TYPE "LBP_typeTMMagazines"
TITLE = Tool management magazines / Almacenes de gestión de herramientas / Magazine zur Werkzeugverwaltung
// User data type to store the magazine data / Tipo de datos de usuario para guardar los datos de almacén / Anwender-Datentyp zum Speichern der Magazindaten
// stored: IsFailsafeCompliant false
   STRUCT
      MaxSpindleNumber : UInt;   // Maximale Spindelanzahl / Maximum spindle number / Número máximo de cabezales
      NumberOfMagazines : UInt;   // Anzahl aller Magazine einschließlich Belade- und Zwischenspeichermagazine / Number of all magazines including loading and buffer magazines / Número total de almacenes, incluidos almacenes de carga e intermedios
      Magazines : Array[1..64] of Struct   // Alle Magazine einschließlich Belade- und Zwischenspeichermagazine / All magazines including loading and buffer magazines / Todos los almacenes, incluidos almacenes de carga e intermedios
         Number : UInt;   // Magazin-Nummer / Magazine number / Número de almacén
         "Type" : UInt;   // Magazintyp / Magazine type / Tipo de almacén
         Places : UInt;   // Anzahl der Plätze im Magazin / Number of locations in magazine / Número de puestos en el almacén
         TMNumber : UInt;   // Werkzeug-Verwaltungsnummer / Tool management number / Número de gestión de herramientas
      END_STRUCT;
   END_STRUCT;
   // // Magazines[2].Number : Magazin-Nummer / Magazine number / Número de almacén
   // // Magazines[3].Number : Magazin-Nummer / Magazine number / Número de almacén
   // // Magazines[4].Number : Magazin-Nummer / Magazine number / Número de almacén
   // // Magazines[5].Number : Magazin-Nummer / Magazine number / Número de almacén
   // // Magazines[6].Number : Magazin-Nummer / Magazine number / Número de almacén
   // // Magazines[7].Number : Magazin-Nummer / Magazine number / Número de almacén
   // // Magazines[8].Number : Magazin-Nummer / Magazine number / Número de almacén
   // // Magazines[9].Number : Magazin-Nummer / Magazine number / Número de almacén
   // // Magazines[10].Number : Magazin-Nummer / Magazine number / Número de almacén
   // // Magazines[11].Number : Magazin-Nummer / Magazine number / Número de almacén
   // // Magazines[12].Number : Magazin-Nummer / Magazine number / Número de almacén
   // // Magazines[13].Number : Magazin-Nummer / Magazine number / Número de almacén
   // // Magazines[14].Number : Magazin-Nummer / Magazine number / Número de almacén
   // // Magazines[15].Number : Magazin-Nummer / Magazine number / Número de almacén
   // // Magazines[16].Number : Magazin-Nummer / Magazine number / Número de almacén
   // // Magazines[17].Number : Magazin-Nummer / Magazine number / Número de almacén
   // // Magazines[18].Number : Magazin-Nummer / Magazine number / Número de almacén
   // // Magazines[19].Number : Magazin-Nummer / Magazine number / Número de almacén
   // // Magazines[20].Number : Magazin-Nummer / Magazine number / Número de almacén
   // // Magazines[21].Number : Magazin-Nummer / Magazine number / Número de almacén
   // // Magazines[22].Number : Magazin-Nummer / Magazine number / Número de almacén
   // // Magazines[23].Number : Magazin-Nummer / Magazine number / Número de almacén
   // // Magazines[24].Number : Magazin-Nummer / Magazine number / Número de almacén
   // // Magazines[25].Number : Magazin-Nummer / Magazine number / Número de almacén
   // // Magazines[26].Number : Magazin-Nummer / Magazine number / Número de almacén
   // // Magazines[27].Number : Magazin-Nummer / Magazine number / Número de almacén
   // // Magazines[28].Number : Magazin-Nummer / Magazine number / Número de almacén
   // // Magazines[29].Number : Magazin-Nummer / Magazine number / Número de almacén
   // // Magazines[30].Number : Magazin-Nummer / Magazine number / Número de almacén
   // // Magazines[31].Number : Magazin-Nummer / Magazine number / Número de almacén
   // // Magazines[32].Number : Magazin-Nummer / Magazine number / Número de almacén
   // // Magazines[33].Number : Magazin-Nummer / Magazine number / Número de almacén
   // // Magazines[34].Number : Magazin-Nummer / Magazine number / Número de almacén
   // // Magazines[35].Number : Magazin-Nummer / Magazine number / Número de almacén
   // // Magazines[36].Number : Magazin-Nummer / Magazine number / Número de almacén
   // // Magazines[37].Number : Magazin-Nummer / Magazine number / Número de almacén
   // // Magazines[38].Number : Magazin-Nummer / Magazine number / Número de almacén
   // // Magazines[39].Number : Magazin-Nummer / Magazine number / Número de almacén
   // // Magazines[40].Number : Magazin-Nummer / Magazine number / Número de almacén
   // // Magazines[41].Number : Magazin-Nummer / Magazine number / Número de almacén
   // // Magazines[42].Number : Magazin-Nummer / Magazine number / Número de almacén
   // // Magazines[43].Number : Magazin-Nummer / Magazine number / Número de almacén
   // // Magazines[44].Number : Magazin-Nummer / Magazine number / Número de almacén
   // // Magazines[45].Number : Magazin-Nummer / Magazine number / Número de almacén
   // // Magazines[46].Number : Magazin-Nummer / Magazine number / Número de almacén
   // // Magazines[47].Number : Magazin-Nummer / Magazine number / Número de almacén
   // // Magazines[48].Number : Magazin-Nummer / Magazine number / Número de almacén
   // // Magazines[49].Number : Magazin-Nummer / Magazine number / Número de almacén
   // // Magazines[50].Number : Magazin-Nummer / Magazine number / Número de almacén
   // // Magazines[51].Number : Magazin-Nummer / Magazine number / Número de almacén
   // // Magazines[52].Number : Magazin-Nummer / Magazine number / Número de almacén
   // // Magazines[53].Number : Magazin-Nummer / Magazine number / Número de almacén
   // // Magazines[54].Number : Magazin-Nummer / Magazine number / Número de almacén
   // // Magazines[55].Number : Magazin-Nummer / Magazine number / Número de almacén
   // // Magazines[56].Number : Magazin-Nummer / Magazine number / Número de almacén
   // // Magazines[57].Number : Magazin-Nummer / Magazine number / Número de almacén
   // // Magazines[58].Number : Magazin-Nummer / Magazine number / Número de almacén
   // // Magazines[59].Number : Magazin-Nummer / Magazine number / Número de almacén
   // // Magazines[60].Number : Magazin-Nummer / Magazine number / Número de almacén
   // // Magazines[61].Number : Magazin-Nummer / Magazine number / Número de almacén
   // // Magazines[62].Number : Magazin-Nummer / Magazine number / Número de almacén
   // // Magazines[63].Number : Magazin-Nummer / Magazine number / Número de almacén
   // // Magazines[64].Number : Magazin-Nummer / Magazine number / Número de almacén
   // // Magazines[2]."Type" : Magazintyp / Magazine type / Tipo de almacén
   // // Magazines[3]."Type" : Magazintyp / Magazine type / Tipo de almacén
   // // Magazines[4]."Type" : Magazintyp / Magazine type / Tipo de almacén
   // // Magazines[5]."Type" : Magazintyp / Magazine type / Tipo de almacén
   // // Magazines[6]."Type" : Magazintyp / Magazine type / Tipo de almacén
   // // Magazines[7]."Type" : Magazintyp / Magazine type / Tipo de almacén
   // // Magazines[8]."Type" : Magazintyp / Magazine type / Tipo de almacén
   // // Magazines[9]."Type" : Magazintyp / Magazine type / Tipo de almacén
   // // Magazines[10]."Type" : Magazintyp / Magazine type / Tipo de almacén
   // // Magazines[11]."Type" : Magazintyp / Magazine type / Tipo de almacén
   // // Magazines[12]."Type" : Magazintyp / Magazine type / Tipo de almacén
   // // Magazines[13]."Type" : Magazintyp / Magazine type / Tipo de almacén
   // // Magazines[14]."Type" : Magazintyp / Magazine type / Tipo de almacén
   // // Magazines[15]."Type" : Magazintyp / Magazine type / Tipo de almacén
   // // Magazines[16]."Type" : Magazintyp / Magazine type / Tipo de almacén
   // // Magazines[17]."Type" : Magazintyp / Magazine type / Tipo de almacén
   // // Magazines[18]."Type" : Magazintyp / Magazine type / Tipo de almacén
   // // Magazines[19]."Type" : Magazintyp / Magazine type / Tipo de almacén
   // // Magazines[20]."Type" : Magazintyp / Magazine type / Tipo de almacén
   // // Magazines[21]."Type" : Magazintyp / Magazine type / Tipo de almacén
   // // Magazines[22]."Type" : Magazintyp / Magazine type / Tipo de almacén
   // // Magazines[23]."Type" : Magazintyp / Magazine type / Tipo de almacén
   // // Magazines[24]."Type" : Magazintyp / Magazine type / Tipo de almacén
   // // Magazines[25]."Type" : Magazintyp / Magazine type / Tipo de almacén
   // // Magazines[26]."Type" : Magazintyp / Magazine type / Tipo de almacén
   // // Magazines[27]."Type" : Magazintyp / Magazine type / Tipo de almacén
   // // Magazines[28]."Type" : Magazintyp / Magazine type / Tipo de almacén
   // // Magazines[29]."Type" : Magazintyp / Magazine type / Tipo de almacén
   // // Magazines[30]."Type" : Magazintyp / Magazine type / Tipo de almacén
   // // Magazines[31]."Type" : Magazintyp / Magazine type / Tipo de almacén
   // // Magazines[32]."Type" : Magazintyp / Magazine type / Tipo de almacén
   // // Magazines[33]."Type" : Magazintyp / Magazine type / Tipo de almacén
   // // Magazines[34]."Type" : Magazintyp / Magazine type / Tipo de almacén
   // // Magazines[35]."Type" : Magazintyp / Magazine type / Tipo de almacén
   // // Magazines[36]."Type" : Magazintyp / Magazine type / Tipo de almacén
   // // Magazines[37]."Type" : Magazintyp / Magazine type / Tipo de almacén
   // // Magazines[38]."Type" : Magazintyp / Magazine type / Tipo de almacén
   // // Magazines[39]."Type" : Magazintyp / Magazine type / Tipo de almacén
   // // Magazines[40]."Type" : Magazintyp / Magazine type / Tipo de almacén
   // // Magazines[41]."Type" : Magazintyp / Magazine type / Tipo de almacén
   // // Magazines[42]."Type" : Magazintyp / Magazine type / Tipo de almacén
   // // Magazines[43]."Type" : Magazintyp / Magazine type / Tipo de almacén
   // // Magazines[44]."Type" : Magazintyp / Magazine type / Tipo de almacén
   // // Magazines[45]."Type" : Magazintyp / Magazine type / Tipo de almacén
   // // Magazines[46]."Type" : Magazintyp / Magazine type / Tipo de almacén
   // // Magazines[47]."Type" : Magazintyp / Magazine type / Tipo de almacén
   // // Magazines[48]."Type" : Magazintyp / Magazine type / Tipo de almacén
   // // Magazines[49]."Type" : Magazintyp / Magazine type / Tipo de almacén
   // // Magazines[50]."Type" : Magazintyp / Magazine type / Tipo de almacén
   // // Magazines[51]."Type" : Magazintyp / Magazine type / Tipo de almacén
   // // Magazines[52]."Type" : Magazintyp / Magazine type / Tipo de almacén
   // // Magazines[53]."Type" : Magazintyp / Magazine type / Tipo de almacén
   // // Magazines[54]."Type" : Magazintyp / Magazine type / Tipo de almacén
   // // Magazines[55]."Type" : Magazintyp / Magazine type / Tipo de almacén
   // // Magazines[56]."Type" : Magazintyp / Magazine type / Tipo de almacén
   // // Magazines[57]."Type" : Magazintyp / Magazine type / Tipo de almacén
   // // Magazines[58]."Type" : Magazintyp / Magazine type / Tipo de almacén
   // // Magazines[59]."Type" : Magazintyp / Magazine type / Tipo de almacén
   // // Magazines[60]."Type" : Magazintyp / Magazine type / Tipo de almacén
   // // Magazines[61]."Type" : Magazintyp / Magazine type / Tipo de almacén
   // // Magazines[62]."Type" : Magazintyp / Magazine type / Tipo de almacén
   // // Magazines[63]."Type" : Magazintyp / Magazine type / Tipo de almacén
   // // Magazines[64]."Type" : Magazintyp / Magazine type / Tipo de almacén
   // // Magazines[2].Places : Anzahl der Plätze im Magazin / Number of locations in magazine / Número de puestos en el almacén
   // // Magazines[3].Places : Anzahl der Plätze im Magazin / Number of locations in magazine / Número de puestos en el almacén
   // // Magazines[4].Places : Anzahl der Plätze im Magazin / Number of locations in magazine / Número de puestos en el almacén
   // // Magazines[5].Places : Anzahl der Plätze im Magazin / Number of locations in magazine / Número de puestos en el almacén
   // // Magazines[6].Places : Anzahl der Plätze im Magazin / Number of locations in magazine / Número de puestos en el almacén
   // // Magazines[7].Places : Anzahl der Plätze im Magazin / Number of locations in magazine / Número de puestos en el almacén
   // // Magazines[8].Places : Anzahl der Plätze im Magazin / Number of locations in magazine / Número de puestos en el almacén
   // // Magazines[9].Places : Anzahl der Plätze im Magazin / Number of locations in magazine / Número de puestos en el almacén
   // // Magazines[10].Places : Anzahl der Plätze im Magazin / Number of locations in magazine / Número de puestos en el almacén
   // // Magazines[11].Places : Anzahl der Plätze im Magazin / Number of locations in magazine / Número de puestos en el almacén
   // // Magazines[12].Places : Anzahl der Plätze im Magazin / Number of locations in magazine / Número de puestos en el almacén
   // // Magazines[13].Places : Anzahl der Plätze im Magazin / Number of locations in magazine / Número de puestos en el almacén
   // // Magazines[14].Places : Anzahl der Plätze im Magazin / Number of locations in magazine / Número de puestos en el almacén
   // // Magazines[15].Places : Anzahl der Plätze im Magazin / Number of locations in magazine / Número de puestos en el almacén
   // // Magazines[16].Places : Anzahl der Plätze im Magazin / Number of locations in magazine / Número de puestos en el almacén
   // // Magazines[17].Places : Anzahl der Plätze im Magazin / Number of locations in magazine / Número de puestos en el almacén
   // // Magazines[18].Places : Anzahl der Plätze im Magazin / Number of locations in magazine / Número de puestos en el almacén
   // // Magazines[19].Places : Anzahl der Plätze im Magazin / Number of locations in magazine / Número de puestos en el almacén
   // // Magazines[20].Places : Anzahl der Plätze im Magazin / Number of locations in magazine / Número de puestos en el almacén
   // // Magazines[21].Places : Anzahl der Plätze im Magazin / Number of locations in magazine / Número de puestos en el almacén
   // // Magazines[22].Places : Anzahl der Plätze im Magazin / Number of locations in magazine / Número de puestos en el almacén
   // // Magazines[23].Places : Anzahl der Plätze im Magazin / Number of locations in magazine / Número de puestos en el almacén
   // // Magazines[24].Places : Anzahl der Plätze im Magazin / Number of locations in magazine / Número de puestos en el almacén
   // // Magazines[25].Places : Anzahl der Plätze im Magazin / Number of locations in magazine / Número de puestos en el almacén
   // // Magazines[26].Places : Anzahl der Plätze im Magazin / Number of locations in magazine / Número de puestos en el almacén
   // // Magazines[27].Places : Anzahl der Plätze im Magazin / Number of locations in magazine / Número de puestos en el almacén
   // // Magazines[28].Places : Anzahl der Plätze im Magazin / Number of locations in magazine / Número de puestos en el almacén
   // // Magazines[29].Places : Anzahl der Plätze im Magazin / Number of locations in magazine / Número de puestos en el almacén
   // // Magazines[30].Places : Anzahl der Plätze im Magazin / Number of locations in magazine / Número de puestos en el almacén
   // // Magazines[31].Places : Anzahl der Plätze im Magazin / Number of locations in magazine / Número de puestos en el almacén
   // // Magazines[32].Places : Anzahl der Plätze im Magazin / Number of locations in magazine / Número de puestos en el almacén
   // // Magazines[33].Places : Anzahl der Plätze im Magazin / Number of locations in magazine / Número de puestos en el almacén
   // // Magazines[34].Places : Anzahl der Plätze im Magazin / Number of locations in magazine / Número de puestos en el almacén
   // // Magazines[35].Places : Anzahl der Plätze im Magazin / Number of locations in magazine / Número de puestos en el almacén
   // // Magazines[36].Places : Anzahl der Plätze im Magazin / Number of locations in magazine / Número de puestos en el almacén
   // // Magazines[37].Places : Anzahl der Plätze im Magazin / Number of locations in magazine / Número de puestos en el almacén
   // // Magazines[38].Places : Anzahl der Plätze im Magazin / Number of locations in magazine / Número de puestos en el almacén
   // // Magazines[39].Places : Anzahl der Plätze im Magazin / Number of locations in magazine / Número de puestos en el almacén
   // // Magazines[40].Places : Anzahl der Plätze im Magazin / Number of locations in magazine / Número de puestos en el almacén
   // // Magazines[41].Places : Anzahl der Plätze im Magazin / Number of locations in magazine / Número de puestos en el almacén
   // // Magazines[42].Places : Anzahl der Plätze im Magazin / Number of locations in magazine / Número de puestos en el almacén
   // // Magazines[43].Places : Anzahl der Plätze im Magazin / Number of locations in magazine / Número de puestos en el almacén
   // // Magazines[44].Places : Anzahl der Plätze im Magazin / Number of locations in magazine / Número de puestos en el almacén
   // // Magazines[45].Places : Anzahl der Plätze im Magazin / Number of locations in magazine / Número de puestos en el almacén
   // // Magazines[46].Places : Anzahl der Plätze im Magazin / Number of locations in magazine / Número de puestos en el almacén
   // // Magazines[47].Places : Anzahl der Plätze im Magazin / Number of locations in magazine / Número de puestos en el almacén
   // // Magazines[48].Places : Anzahl der Plätze im Magazin / Number of locations in magazine / Número de puestos en el almacén
   // // Magazines[49].Places : Anzahl der Plätze im Magazin / Number of locations in magazine / Número de puestos en el almacén
   // // Magazines[50].Places : Anzahl der Plätze im Magazin / Number of locations in magazine / Número de puestos en el almacén
   // // Magazines[51].Places : Anzahl der Plätze im Magazin / Number of locations in magazine / Número de puestos en el almacén
   // // Magazines[52].Places : Anzahl der Plätze im Magazin / Number of locations in magazine / Número de puestos en el almacén
   // // Magazines[53].Places : Anzahl der Plätze im Magazin / Number of locations in magazine / Número de puestos en el almacén
   // // Magazines[54].Places : Anzahl der Plätze im Magazin / Number of locations in magazine / Número de puestos en el almacén
   // // Magazines[55].Places : Anzahl der Plätze im Magazin / Number of locations in magazine / Número de puestos en el almacén
   // // Magazines[56].Places : Anzahl der Plätze im Magazin / Number of locations in magazine / Número de puestos en el almacén
   // // Magazines[57].Places : Anzahl der Plätze im Magazin / Number of locations in magazine / Número de puestos en el almacén
   // // Magazines[58].Places : Anzahl der Plätze im Magazin / Number of locations in magazine / Número de puestos en el almacén
   // // Magazines[59].Places : Anzahl der Plätze im Magazin / Number of locations in magazine / Número de puestos en el almacén
   // // Magazines[60].Places : Anzahl der Plätze im Magazin / Number of locations in magazine / Número de puestos en el almacén
   // // Magazines[61].Places : Anzahl der Plätze im Magazin / Number of locations in magazine / Número de puestos en el almacén
   // // Magazines[62].Places : Anzahl der Plätze im Magazin / Number of locations in magazine / Número de puestos en el almacén
   // // Magazines[63].Places : Anzahl der Plätze im Magazin / Number of locations in magazine / Número de puestos en el almacén
   // // Magazines[64].Places : Anzahl der Plätze im Magazin / Number of locations in magazine / Número de puestos en el almacén
   // // Magazines[2].TMNumber : Werkzeug-Verwaltungsnummer / Tool management number / Número de gestión de herramientas
   // // Magazines[3].TMNumber : Werkzeug-Verwaltungsnummer / Tool management number / Número de gestión de herramientas
   // // Magazines[4].TMNumber : Werkzeug-Verwaltungsnummer / Tool management number / Número de gestión de herramientas
   // // Magazines[5].TMNumber : Werkzeug-Verwaltungsnummer / Tool management number / Número de gestión de herramientas
   // // Magazines[6].TMNumber : Werkzeug-Verwaltungsnummer / Tool management number / Número de gestión de herramientas
   // // Magazines[7].TMNumber : Werkzeug-Verwaltungsnummer / Tool management number / Número de gestión de herramientas
   // // Magazines[8].TMNumber : Werkzeug-Verwaltungsnummer / Tool management number / Número de gestión de herramientas
   // // Magazines[9].TMNumber : Werkzeug-Verwaltungsnummer / Tool management number / Número de gestión de herramientas
   // // Magazines[10].TMNumber : Werkzeug-Verwaltungsnummer / Tool management number / Número de gestión de herramientas
   // // Magazines[11].TMNumber : Werkzeug-Verwaltungsnummer / Tool management number / Número de gestión de herramientas
   // // Magazines[12].TMNumber : Werkzeug-Verwaltungsnummer / Tool management number / Número de gestión de herramientas
   // // Magazines[13].TMNumber : Werkzeug-Verwaltungsnummer / Tool management number / Número de gestión de herramientas
   // // Magazines[14].TMNumber : Werkzeug-Verwaltungsnummer / Tool management number / Número de gestión de herramientas
   // // Magazines[15].TMNumber : Werkzeug-Verwaltungsnummer / Tool management number / Número de gestión de herramientas
   // // Magazines[16].TMNumber : Werkzeug-Verwaltungsnummer / Tool management number / Número de gestión de herramientas
   // // Magazines[17].TMNumber : Werkzeug-Verwaltungsnummer / Tool management number / Número de gestión de herramientas
   // // Magazines[18].TMNumber : Werkzeug-Verwaltungsnummer / Tool management number / Número de gestión de herramientas
   // // Magazines[19].TMNumber : Werkzeug-Verwaltungsnummer / Tool management number / Número de gestión de herramientas
   // // Magazines[20].TMNumber : Werkzeug-Verwaltungsnummer / Tool management number / Número de gestión de herramientas
   // // Magazines[21].TMNumber : Werkzeug-Verwaltungsnummer / Tool management number / Número de gestión de herramientas
   // // Magazines[22].TMNumber : Werkzeug-Verwaltungsnummer / Tool management number / Número de gestión de herramientas
   // // Magazines[23].TMNumber : Werkzeug-Verwaltungsnummer / Tool management number / Número de gestión de herramientas
   // // Magazines[24].TMNumber : Werkzeug-Verwaltungsnummer / Tool management number / Número de gestión de herramientas
   // // Magazines[25].TMNumber : Werkzeug-Verwaltungsnummer / Tool management number / Número de gestión de herramientas
   // // Magazines[26].TMNumber : Werkzeug-Verwaltungsnummer / Tool management number / Número de gestión de herramientas
   // // Magazines[27].TMNumber : Werkzeug-Verwaltungsnummer / Tool management number / Número de gestión de herramientas
   // // Magazines[28].TMNumber : Werkzeug-Verwaltungsnummer / Tool management number / Número de gestión de herramientas
   // // Magazines[29].TMNumber : Werkzeug-Verwaltungsnummer / Tool management number / Número de gestión de herramientas
   // // Magazines[30].TMNumber : Werkzeug-Verwaltungsnummer / Tool management number / Número de gestión de herramientas
   // // Magazines[31].TMNumber : Werkzeug-Verwaltungsnummer / Tool management number / Número de gestión de herramientas
   // // Magazines[32].TMNumber : Werkzeug-Verwaltungsnummer / Tool management number / Número de gestión de herramientas
   // // Magazines[33].TMNumber : Werkzeug-Verwaltungsnummer / Tool management number / Número de gestión de herramientas
   // // Magazines[34].TMNumber : Werkzeug-Verwaltungsnummer / Tool management number / Número de gestión de herramientas
   // // Magazines[35].TMNumber : Werkzeug-Verwaltungsnummer / Tool management number / Número de gestión de herramientas
   // // Magazines[36].TMNumber : Werkzeug-Verwaltungsnummer / Tool management number / Número de gestión de herramientas
   // // Magazines[37].TMNumber : Werkzeug-Verwaltungsnummer / Tool management number / Número de gestión de herramientas
   // // Magazines[38].TMNumber : Werkzeug-Verwaltungsnummer / Tool management number / Número de gestión de herramientas
   // // Magazines[39].TMNumber : Werkzeug-Verwaltungsnummer / Tool management number / Número de gestión de herramientas
   // // Magazines[40].TMNumber : Werkzeug-Verwaltungsnummer / Tool management number / Número de gestión de herramientas
   // // Magazines[41].TMNumber : Werkzeug-Verwaltungsnummer / Tool management number / Número de gestión de herramientas
   // // Magazines[42].TMNumber : Werkzeug-Verwaltungsnummer / Tool management number / Número de gestión de herramientas
   // // Magazines[43].TMNumber : Werkzeug-Verwaltungsnummer / Tool management number / Número de gestión de herramientas
   // // Magazines[44].TMNumber : Werkzeug-Verwaltungsnummer / Tool management number / Número de gestión de herramientas
   // // Magazines[45].TMNumber : Werkzeug-Verwaltungsnummer / Tool management number / Número de gestión de herramientas
   // // Magazines[46].TMNumber : Werkzeug-Verwaltungsnummer / Tool management number / Número de gestión de herramientas
   // // Magazines[47].TMNumber : Werkzeug-Verwaltungsnummer / Tool management number / Número de gestión de herramientas
   // // Magazines[48].TMNumber : Werkzeug-Verwaltungsnummer / Tool management number / Número de gestión de herramientas
   // // Magazines[49].TMNumber : Werkzeug-Verwaltungsnummer / Tool management number / Número de gestión de herramientas
   // // Magazines[50].TMNumber : Werkzeug-Verwaltungsnummer / Tool management number / Número de gestión de herramientas
   // // Magazines[51].TMNumber : Werkzeug-Verwaltungsnummer / Tool management number / Número de gestión de herramientas
   // // Magazines[52].TMNumber : Werkzeug-Verwaltungsnummer / Tool management number / Número de gestión de herramientas
   // // Magazines[53].TMNumber : Werkzeug-Verwaltungsnummer / Tool management number / Número de gestión de herramientas
   // // Magazines[54].TMNumber : Werkzeug-Verwaltungsnummer / Tool management number / Número de gestión de herramientas
   // // Magazines[55].TMNumber : Werkzeug-Verwaltungsnummer / Tool management number / Número de gestión de herramientas
   // // Magazines[56].TMNumber : Werkzeug-Verwaltungsnummer / Tool management number / Número de gestión de herramientas
   // // Magazines[57].TMNumber : Werkzeug-Verwaltungsnummer / Tool management number / Número de gestión de herramientas
   // // Magazines[58].TMNumber : Werkzeug-Verwaltungsnummer / Tool management number / Número de gestión de herramientas
   // // Magazines[59].TMNumber : Werkzeug-Verwaltungsnummer / Tool management number / Número de gestión de herramientas
   // // Magazines[60].TMNumber : Werkzeug-Verwaltungsnummer / Tool management number / Número de gestión de herramientas
   // // Magazines[61].TMNumber : Werkzeug-Verwaltungsnummer / Tool management number / Número de gestión de herramientas
   // // Magazines[62].TMNumber : Werkzeug-Verwaltungsnummer / Tool management number / Número de gestión de herramientas
   // // Magazines[63].TMNumber : Werkzeug-Verwaltungsnummer / Tool management number / Número de gestión de herramientas
   // // Magazines[64].TMNumber : Werkzeug-Verwaltungsnummer / Tool management number / Número de gestión de herramientas
   // // Magazines[1] : Alle Magazine einschließlich Belade- und Zwischenspeichermagazine / All magazines including loading and buffer magazines / Todos los almacenes, incluidos almacenes de carga e intermedios
   // // Magazines[2] : Alle Magazine einschließlich Belade- und Zwischenspeichermagazine / All magazines including loading and buffer magazines / Todos los almacenes, incluidos almacenes de carga e intermedios
   // // Magazines[3] : Alle Magazine einschließlich Belade- und Zwischenspeichermagazine / All magazines including loading and buffer magazines / Todos los almacenes, incluidos almacenes de carga e intermedios
   // // Magazines[4] : Alle Magazine einschließlich Belade- und Zwischenspeichermagazine / All magazines including loading and buffer magazines / Todos los almacenes, incluidos almacenes de carga e intermedios
   // // Magazines[5] : Alle Magazine einschließlich Belade- und Zwischenspeichermagazine / All magazines including loading and buffer magazines / Todos los almacenes, incluidos almacenes de carga e intermedios
   // // Magazines[6] : Alle Magazine einschließlich Belade- und Zwischenspeichermagazine / All magazines including loading and buffer magazines / Todos los almacenes, incluidos almacenes de carga e intermedios
   // // Magazines[7] : Alle Magazine einschließlich Belade- und Zwischenspeichermagazine / All magazines including loading and buffer magazines / Todos los almacenes, incluidos almacenes de carga e intermedios
   // // Magazines[8] : Alle Magazine einschließlich Belade- und Zwischenspeichermagazine / All magazines including loading and buffer magazines / Todos los almacenes, incluidos almacenes de carga e intermedios
   // // Magazines[9] : Alle Magazine einschließlich Belade- und Zwischenspeichermagazine / All magazines including loading and buffer magazines / Todos los almacenes, incluidos almacenes de carga e intermedios
   // // Magazines[10] : Alle Magazine einschließlich Belade- und Zwischenspeichermagazine / All magazines including loading and buffer magazines / Todos los almacenes, incluidos almacenes de carga e intermedios
   // // Magazines[11] : Alle Magazine einschließlich Belade- und Zwischenspeichermagazine / All magazines including loading and buffer magazines / Todos los almacenes, incluidos almacenes de carga e intermedios
   // // Magazines[12] : Alle Magazine einschließlich Belade- und Zwischenspeichermagazine / All magazines including loading and buffer magazines / Todos los almacenes, incluidos almacenes de carga e intermedios
   // // Magazines[13] : Alle Magazine einschließlich Belade- und Zwischenspeichermagazine / All magazines including loading and buffer magazines / Todos los almacenes, incluidos almacenes de carga e intermedios
   // // Magazines[14] : Alle Magazine einschließlich Belade- und Zwischenspeichermagazine / All magazines including loading and buffer magazines / Todos los almacenes, incluidos almacenes de carga e intermedios
   // // Magazines[15] : Alle Magazine einschließlich Belade- und Zwischenspeichermagazine / All magazines including loading and buffer magazines / Todos los almacenes, incluidos almacenes de carga e intermedios
   // // Magazines[16] : Alle Magazine einschließlich Belade- und Zwischenspeichermagazine / All magazines including loading and buffer magazines / Todos los almacenes, incluidos almacenes de carga e intermedios
   // // Magazines[17] : Alle Magazine einschließlich Belade- und Zwischenspeichermagazine / All magazines including loading and buffer magazines / Todos los almacenes, incluidos almacenes de carga e intermedios
   // // Magazines[18] : Alle Magazine einschließlich Belade- und Zwischenspeichermagazine / All magazines including loading and buffer magazines / Todos los almacenes, incluidos almacenes de carga e intermedios
   // // Magazines[19] : Alle Magazine einschließlich Belade- und Zwischenspeichermagazine / All magazines including loading and buffer magazines / Todos los almacenes, incluidos almacenes de carga e intermedios
   // // Magazines[20] : Alle Magazine einschließlich Belade- und Zwischenspeichermagazine / All magazines including loading and buffer magazines / Todos los almacenes, incluidos almacenes de carga e intermedios
   // // Magazines[21] : Alle Magazine einschließlich Belade- und Zwischenspeichermagazine / All magazines including loading and buffer magazines / Todos los almacenes, incluidos almacenes de carga e intermedios
   // // Magazines[22] : Alle Magazine einschließlich Belade- und Zwischenspeichermagazine / All magazines including loading and buffer magazines / Todos los almacenes, incluidos almacenes de carga e intermedios
   // // Magazines[23] : Alle Magazine einschließlich Belade- und Zwischenspeichermagazine / All magazines including loading and buffer magazines / Todos los almacenes, incluidos almacenes de carga e intermedios
   // // Magazines[24] : Alle Magazine einschließlich Belade- und Zwischenspeichermagazine / All magazines including loading and buffer magazines / Todos los almacenes, incluidos almacenes de carga e intermedios
   // // Magazines[25] : Alle Magazine einschließlich Belade- und Zwischenspeichermagazine / All magazines including loading and buffer magazines / Todos los almacenes, incluidos almacenes de carga e intermedios
   // // Magazines[26] : Alle Magazine einschließlich Belade- und Zwischenspeichermagazine / All magazines including loading and buffer magazines / Todos los almacenes, incluidos almacenes de carga e intermedios
   // // Magazines[27] : Alle Magazine einschließlich Belade- und Zwischenspeichermagazine / All magazines including loading and buffer magazines / Todos los almacenes, incluidos almacenes de carga e intermedios
   // // Magazines[28] : Alle Magazine einschließlich Belade- und Zwischenspeichermagazine / All magazines including loading and buffer magazines / Todos los almacenes, incluidos almacenes de carga e intermedios
   // // Magazines[29] : Alle Magazine einschließlich Belade- und Zwischenspeichermagazine / All magazines including loading and buffer magazines / Todos los almacenes, incluidos almacenes de carga e intermedios
   // // Magazines[30] : Alle Magazine einschließlich Belade- und Zwischenspeichermagazine / All magazines including loading and buffer magazines / Todos los almacenes, incluidos almacenes de carga e intermedios
   // // Magazines[31] : Alle Magazine einschließlich Belade- und Zwischenspeichermagazine / All magazines including loading and buffer magazines / Todos los almacenes, incluidos almacenes de carga e intermedios
   // // Magazines[32] : Alle Magazine einschließlich Belade- und Zwischenspeichermagazine / All magazines including loading and buffer magazines / Todos los almacenes, incluidos almacenes de carga e intermedios
   // // Magazines[33] : Alle Magazine einschließlich Belade- und Zwischenspeichermagazine / All magazines including loading and buffer magazines / Todos los almacenes, incluidos almacenes de carga e intermedios
   // // Magazines[34] : Alle Magazine einschließlich Belade- und Zwischenspeichermagazine / All magazines including loading and buffer magazines / Todos los almacenes, incluidos almacenes de carga e intermedios
   // // Magazines[35] : Alle Magazine einschließlich Belade- und Zwischenspeichermagazine / All magazines including loading and buffer magazines / Todos los almacenes, incluidos almacenes de carga e intermedios
   // // Magazines[36] : Alle Magazine einschließlich Belade- und Zwischenspeichermagazine / All magazines including loading and buffer magazines / Todos los almacenes, incluidos almacenes de carga e intermedios
   // // Magazines[37] : Alle Magazine einschließlich Belade- und Zwischenspeichermagazine / All magazines including loading and buffer magazines / Todos los almacenes, incluidos almacenes de carga e intermedios
   // // Magazines[38] : Alle Magazine einschließlich Belade- und Zwischenspeichermagazine / All magazines including loading and buffer magazines / Todos los almacenes, incluidos almacenes de carga e intermedios
   // // Magazines[39] : Alle Magazine einschließlich Belade- und Zwischenspeichermagazine / All magazines including loading and buffer magazines / Todos los almacenes, incluidos almacenes de carga e intermedios
   // // Magazines[40] : Alle Magazine einschließlich Belade- und Zwischenspeichermagazine / All magazines including loading and buffer magazines / Todos los almacenes, incluidos almacenes de carga e intermedios
   // // Magazines[41] : Alle Magazine einschließlich Belade- und Zwischenspeichermagazine / All magazines including loading and buffer magazines / Todos los almacenes, incluidos almacenes de carga e intermedios
   // // Magazines[42] : Alle Magazine einschließlich Belade- und Zwischenspeichermagazine / All magazines including loading and buffer magazines / Todos los almacenes, incluidos almacenes de carga e intermedios
   // // Magazines[43] : Alle Magazine einschließlich Belade- und Zwischenspeichermagazine / All magazines including loading and buffer magazines / Todos los almacenes, incluidos almacenes de carga e intermedios
   // // Magazines[44] : Alle Magazine einschließlich Belade- und Zwischenspeichermagazine / All magazines including loading and buffer magazines / Todos los almacenes, incluidos almacenes de carga e intermedios
   // // Magazines[45] : Alle Magazine einschließlich Belade- und Zwischenspeichermagazine / All magazines including loading and buffer magazines / Todos los almacenes, incluidos almacenes de carga e intermedios
   // // Magazines[46] : Alle Magazine einschließlich Belade- und Zwischenspeichermagazine / All magazines including loading and buffer magazines / Todos los almacenes, incluidos almacenes de carga e intermedios
   // // Magazines[47] : Alle Magazine einschließlich Belade- und Zwischenspeichermagazine / All magazines including loading and buffer magazines / Todos los almacenes, incluidos almacenes de carga e intermedios
   // // Magazines[48] : Alle Magazine einschließlich Belade- und Zwischenspeichermagazine / All magazines including loading and buffer magazines / Todos los almacenes, incluidos almacenes de carga e intermedios
   // // Magazines[49] : Alle Magazine einschließlich Belade- und Zwischenspeichermagazine / All magazines including loading and buffer magazines / Todos los almacenes, incluidos almacenes de carga e intermedios
   // // Magazines[50] : Alle Magazine einschließlich Belade- und Zwischenspeichermagazine / All magazines including loading and buffer magazines / Todos los almacenes, incluidos almacenes de carga e intermedios
   // // Magazines[51] : Alle Magazine einschließlich Belade- und Zwischenspeichermagazine / All magazines including loading and buffer magazines / Todos los almacenes, incluidos almacenes de carga e intermedios
   // // Magazines[52] : Alle Magazine einschließlich Belade- und Zwischenspeichermagazine / All magazines including loading and buffer magazines / Todos los almacenes, incluidos almacenes de carga e intermedios
   // // Magazines[53] : Alle Magazine einschließlich Belade- und Zwischenspeichermagazine / All magazines including loading and buffer magazines / Todos los almacenes, incluidos almacenes de carga e intermedios
   // // Magazines[54] : Alle Magazine einschließlich Belade- und Zwischenspeichermagazine / All magazines including loading and buffer magazines / Todos los almacenes, incluidos almacenes de carga e intermedios
   // // Magazines[55] : Alle Magazine einschließlich Belade- und Zwischenspeichermagazine / All magazines including loading and buffer magazines / Todos los almacenes, incluidos almacenes de carga e intermedios
   // // Magazines[56] : Alle Magazine einschließlich Belade- und Zwischenspeichermagazine / All magazines including loading and buffer magazines / Todos los almacenes, incluidos almacenes de carga e intermedios
   // // Magazines[57] : Alle Magazine einschließlich Belade- und Zwischenspeichermagazine / All magazines including loading and buffer magazines / Todos los almacenes, incluidos almacenes de carga e intermedios
   // // Magazines[58] : Alle Magazine einschließlich Belade- und Zwischenspeichermagazine / All magazines including loading and buffer magazines / Todos los almacenes, incluidos almacenes de carga e intermedios
   // // Magazines[59] : Alle Magazine einschließlich Belade- und Zwischenspeichermagazine / All magazines including loading and buffer magazines / Todos los almacenes, incluidos almacenes de carga e intermedios
   // // Magazines[60] : Alle Magazine einschließlich Belade- und Zwischenspeichermagazine / All magazines including loading and buffer magazines / Todos los almacenes, incluidos almacenes de carga e intermedios
   // // Magazines[61] : Alle Magazine einschließlich Belade- und Zwischenspeichermagazine / All magazines including loading and buffer magazines / Todos los almacenes, incluidos almacenes de carga e intermedios
   // // Magazines[62] : Alle Magazine einschließlich Belade- und Zwischenspeichermagazine / All magazines including loading and buffer magazines / Todos los almacenes, incluidos almacenes de carga e intermedios
   // // Magazines[63] : Alle Magazine einschließlich Belade- und Zwischenspeichermagazine / All magazines including loading and buffer magazines / Todos los almacenes, incluidos almacenes de carga e intermedios
   // // Magazines[64] : Alle Magazine einschließlich Belade- und Zwischenspeichermagazine / All magazines including loading and buffer magazines / Todos los almacenes, incluidos almacenes de carga e intermedios
END_TYPE

TYPE "LBP_typeTMSpindle"
TITLE = Tool management / Gestión de herramientas / Werkzeugverwaltung
// User data type for block LBP_TMSpindle [DB72] / Tipo de dato de usuario para bloque LBP_TMSpindle [DB72] / Anwender-Datentyp für Baustein LBP_TMSpindle [DB72]
// stored: IsFailsafeCompliant false
   STRUCT
      IFNo : Array[1..16] of Bool;   // Schnittstelle [Nummer] aktiv / Interface [number] active / Interfaz [número] activa
      Quit : Array[1..16] of Bool;   // Quit-End durchführen / Perform Quit-End / Ejecutar Finalizar confirmación
      TIF : Array[1..16] of Struct
         Comp : Bool;   // Obligatorische Änderung / Compulsory change / Cambio obligatorio
         Perform : Bool;   // Änderung/Wechsel durchführen / Perform change / Ejecutar cambio
         Prepare : Bool;   // Änderung/Wechsel vorbereiten / Prepare change / Preparar cambio
         T0 : Bool;   // T0 programmiert / T0 programmed / T0 programado
         OldTinDBW42 : Bool;   // Puffernummer des vorherigen Werkzeugs in DBW (n+42) / Buffer number of previous tool in DBW (n+42) / Número de búfer de la herramienta previa en DBW (n+42)
         ManTIn : Bool;   // Handwerkzeug manuell in Spindel laden / Load hand tool in spindle manually / Cargar a mano herramienta manual en cabezal
         ManTOut : Bool;   // Handwerkzeug manuell aus Spindel entladen / Unload hand tool from spindle manually / Descargar a mano herramienta manual del cabezal
         SpiTRSpi : Bool;   // Spindelwerkzeug verbleibt in der Spindel / Spindle tool remains in spindle / Herramienta del cabezal permanece en el cabezal
         PerfStatusError : Bool;   // Negative Quittung / Negative acknowledge / Confirmación negativa
         n1_1 : Bool;   // Reserviert / Reserved / Reservado
         n1_2 : Bool;   // Reserviert / Reserved / Reservado
         n1_3 : Bool;   // Reserviert / Reserved / Reservado
         n1_4 : Bool;   // Reserviert / Reserved / Reservado
         n1_5 : Bool;   // Reserviert / Reserved / Reservado
         n1_6 : Bool;   // Reserviert / Reserved / Reservado
         DataInDB1072 : Bool;   // Multitool-Daten gespeichert in DB1072 / Multitool data stored in DB1072 / Datos Multitool guardados en DB1072
         Channel : Byte;   // Zugeordneter Kanal / Assigned channel / Canal asignado
         TMNo : Byte;   // Werkzeug-Verwaltungsnummer / Tool management number / Número de gestión de herramientas
         VdiTcp0 : DInt;   // Freie Anwendervariable 0 / User parameter 0 / Parámetro de usuario 0
         VdiTcp1 : DInt;   // Freie Anwendervariable 1 / User parameter 1 / Parámetro de usuario 1
         VdiTcp2 : DInt;   // Freie Anwendervariable 2 / User parameter 2 / Parámetro de usuario 2
         BufferIdent : Int;   // Puffer-Identifikation (Festwert 9998) / Buffer identification (fixed value 9998) / Identificación de búfer (valor fijo 9998)
         BufferNo : Int;   // Relativer Platz (Ziel) im Puffer / Relative location (target) in the buffer / Puesto relativo (destino) en el búfer
         SMag : Int;   // Magazin-Nummer (Quelle) für neues Werkzeug / Magazine number (source) for new tool / Número de almacén (origen) para nueva herramienta
         SLoc : Int;   // Platznummer (Quelle) für neues Werkzeug / Location number (source) for new tool / Número de puesto (origen) para nueva herramienta
         TMag : Int;   // Magazin-Nummer (Ziel) für vorheriges Werkzeug / Magazine number (target) for previous tool / Número de almacén (destino) para herramienta previa
         TLoc : Int;   // Platznummer (Ziel) für vorheriges Werkzeug / Location number (target) for previous tool / Número de puesto (destino) para herramienta previa
         LocType : Int;   // Werkzeug neu: Platzart / Tool new: location type / Herramienta nueva: tipo de puesto
         SLeft : Int;   // Werkeug neu: Größe links / Tool new: size left / Herramienta nueva: tamaño izquierda
         SRight : Int;   // Werkeug neu: Größe rechts / Tool new: size right / Herramienta nueva: tamaño derecha
         STop : Int;   // Werkeug neu: Größe oben / Tool new: size top / Herramienta nueva: tamaño arriba
         SBottom : Int;   // Werkeug neu: Größe unten / Tool new: size bottom / Herramienta nueva: tamaño abajo
         TInBuffer : Bool;   // ID für Werkzeuge im Puffer / ID for tools in buffer / ID para herramientas en búfer
         IgnoreDisabled : Bool;   // Deaktiviert ignorieren / Ignore disabled / Ignorar desactivado
         Unload : Bool;   // Zu entladen / To be unloaded / Por descargar
         Load : Bool;   // Zu laden / To be loaded / Por cargar
         MasterTool : Bool;   // Master-Werkzeug / Master tool / Herramienta maestra
         n38_5 : Bool;   // Reserviert / Reserved / Reservado
         Exchange_1to1 : Bool;   // 1:1 Austausch / 1:1 exchange / Cambio 1:1
         HandTool : Bool;   // Handwerkzeug / Hand tool / Herramienta manual
         Active : Bool;   // Aktives Werkzeug / Active tool / Herramienta activa
         Enabled : Bool;   // Werkzeug aktiviert / Tool enabled / Herramienta activada
         Disabled : Bool;   // Werkzeug deaktiviert / Tool disabled / Herramienta desactivada
         Measured : Bool;   // Werkzeug gemessen / Tool measured / Herramienta medida
         Prewarn : Bool;   // Vorwarnungsgrenze erreicht / Prewarning limit reached / Límite de prealarma alcanzado
         Change : Bool;   // Werkzeug wird gewechselt / Tool being changed / Sustituyendo herramienta
         FixedLoc : Bool;   // Werkzeug-Festplatz codiert / Tool fixed location coded / Puesto fijo de herramienta codificado
         Used : Bool;   // Werkzeug war in Gebrauch / Tool was in use / La herramienta estaba en uso
         TNo : Int;   // Werkzeug neu: WZ-Nummer / Tool new: T number / Herramienta nueva: n.º herramienta
         OldTBufferNo : Int;   // Puffernummer des vorherigen Werkzeugs / Buffer number of previous tool / Número de búfer de la herramienta previa
         MyMag : Int;   // Originalmagazin des neuen Werkzeugs / Original magazine of new tool / Almacén de origen de la nueva herramienta
         MyPlace : Int;   // Originalplatz des neuen Werkzeugs / Original location of new tool / Puesto de origen de la nueva herramienta
      END_STRUCT;
   END_STRUCT;
   // // TIF[2].Comp : Obligatorische Änderung / Compulsory change / Cambio obligatorio
   // // TIF[3].Comp : Obligatorische Änderung / Compulsory change / Cambio obligatorio
   // // TIF[4].Comp : Obligatorische Änderung / Compulsory change / Cambio obligatorio
   // // TIF[5].Comp : Obligatorische Änderung / Compulsory change / Cambio obligatorio
   // // TIF[6].Comp : Obligatorische Änderung / Compulsory change / Cambio obligatorio
   // // TIF[7].Comp : Obligatorische Änderung / Compulsory change / Cambio obligatorio
   // // TIF[8].Comp : Obligatorische Änderung / Compulsory change / Cambio obligatorio
   // // TIF[9].Comp : Obligatorische Änderung / Compulsory change / Cambio obligatorio
   // // TIF[10].Comp : Obligatorische Änderung / Compulsory change / Cambio obligatorio
   // // TIF[11].Comp : Obligatorische Änderung / Compulsory change / Cambio obligatorio
   // // TIF[12].Comp : Obligatorische Änderung / Compulsory change / Cambio obligatorio
   // // TIF[13].Comp : Obligatorische Änderung / Compulsory change / Cambio obligatorio
   // // TIF[14].Comp : Obligatorische Änderung / Compulsory change / Cambio obligatorio
   // // TIF[15].Comp : Obligatorische Änderung / Compulsory change / Cambio obligatorio
   // // TIF[16].Comp : Obligatorische Änderung / Compulsory change / Cambio obligatorio
   // // TIF[2].Perform : Änderung/Wechsel durchführen / Perform change / Ejecutar cambio
   // // TIF[3].Perform : Änderung/Wechsel durchführen / Perform change / Ejecutar cambio
   // // TIF[4].Perform : Änderung/Wechsel durchführen / Perform change / Ejecutar cambio
   // // TIF[5].Perform : Änderung/Wechsel durchführen / Perform change / Ejecutar cambio
   // // TIF[6].Perform : Änderung/Wechsel durchführen / Perform change / Ejecutar cambio
   // // TIF[7].Perform : Änderung/Wechsel durchführen / Perform change / Ejecutar cambio
   // // TIF[8].Perform : Änderung/Wechsel durchführen / Perform change / Ejecutar cambio
   // // TIF[9].Perform : Änderung/Wechsel durchführen / Perform change / Ejecutar cambio
   // // TIF[10].Perform : Änderung/Wechsel durchführen / Perform change / Ejecutar cambio
   // // TIF[11].Perform : Änderung/Wechsel durchführen / Perform change / Ejecutar cambio
   // // TIF[12].Perform : Änderung/Wechsel durchführen / Perform change / Ejecutar cambio
   // // TIF[13].Perform : Änderung/Wechsel durchführen / Perform change / Ejecutar cambio
   // // TIF[14].Perform : Änderung/Wechsel durchführen / Perform change / Ejecutar cambio
   // // TIF[15].Perform : Änderung/Wechsel durchführen / Perform change / Ejecutar cambio
   // // TIF[16].Perform : Änderung/Wechsel durchführen / Perform change / Ejecutar cambio
   // // TIF[2].Prepare : Änderung/Wechsel vorbereiten / Prepare change / Preparar cambio
   // // TIF[3].Prepare : Änderung/Wechsel vorbereiten / Prepare change / Preparar cambio
   // // TIF[4].Prepare : Änderung/Wechsel vorbereiten / Prepare change / Preparar cambio
   // // TIF[5].Prepare : Änderung/Wechsel vorbereiten / Prepare change / Preparar cambio
   // // TIF[6].Prepare : Änderung/Wechsel vorbereiten / Prepare change / Preparar cambio
   // // TIF[7].Prepare : Änderung/Wechsel vorbereiten / Prepare change / Preparar cambio
   // // TIF[8].Prepare : Änderung/Wechsel vorbereiten / Prepare change / Preparar cambio
   // // TIF[9].Prepare : Änderung/Wechsel vorbereiten / Prepare change / Preparar cambio
   // // TIF[10].Prepare : Änderung/Wechsel vorbereiten / Prepare change / Preparar cambio
   // // TIF[11].Prepare : Änderung/Wechsel vorbereiten / Prepare change / Preparar cambio
   // // TIF[12].Prepare : Änderung/Wechsel vorbereiten / Prepare change / Preparar cambio
   // // TIF[13].Prepare : Änderung/Wechsel vorbereiten / Prepare change / Preparar cambio
   // // TIF[14].Prepare : Änderung/Wechsel vorbereiten / Prepare change / Preparar cambio
   // // TIF[15].Prepare : Änderung/Wechsel vorbereiten / Prepare change / Preparar cambio
   // // TIF[16].Prepare : Änderung/Wechsel vorbereiten / Prepare change / Preparar cambio
   // // TIF[2].T0 : T0 programmiert / T0 programmed / T0 programado
   // // TIF[3].T0 : T0 programmiert / T0 programmed / T0 programado
   // // TIF[4].T0 : T0 programmiert / T0 programmed / T0 programado
   // // TIF[5].T0 : T0 programmiert / T0 programmed / T0 programado
   // // TIF[6].T0 : T0 programmiert / T0 programmed / T0 programado
   // // TIF[7].T0 : T0 programmiert / T0 programmed / T0 programado
   // // TIF[8].T0 : T0 programmiert / T0 programmed / T0 programado
   // // TIF[9].T0 : T0 programmiert / T0 programmed / T0 programado
   // // TIF[10].T0 : T0 programmiert / T0 programmed / T0 programado
   // // TIF[11].T0 : T0 programmiert / T0 programmed / T0 programado
   // // TIF[12].T0 : T0 programmiert / T0 programmed / T0 programado
   // // TIF[13].T0 : T0 programmiert / T0 programmed / T0 programado
   // // TIF[14].T0 : T0 programmiert / T0 programmed / T0 programado
   // // TIF[15].T0 : T0 programmiert / T0 programmed / T0 programado
   // // TIF[16].T0 : T0 programmiert / T0 programmed / T0 programado
   // // TIF[2].OldTinDBW42 : Puffernummer des vorherigen Werkzeugs in DBW (n+42) / Buffer number of previous tool in DBW (n+42) / Número de búfer de la herramienta previa en DBW (n+42)
   // // TIF[3].OldTinDBW42 : Puffernummer des vorherigen Werkzeugs in DBW (n+42) / Buffer number of previous tool in DBW (n+42) / Número de búfer de la herramienta previa en DBW (n+42)
   // // TIF[4].OldTinDBW42 : Puffernummer des vorherigen Werkzeugs in DBW (n+42) / Buffer number of previous tool in DBW (n+42) / Número de búfer de la herramienta previa en DBW (n+42)
   // // TIF[5].OldTinDBW42 : Puffernummer des vorherigen Werkzeugs in DBW (n+42) / Buffer number of previous tool in DBW (n+42) / Número de búfer de la herramienta previa en DBW (n+42)
   // // TIF[6].OldTinDBW42 : Puffernummer des vorherigen Werkzeugs in DBW (n+42) / Buffer number of previous tool in DBW (n+42) / Número de búfer de la herramienta previa en DBW (n+42)
   // // TIF[7].OldTinDBW42 : Puffernummer des vorherigen Werkzeugs in DBW (n+42) / Buffer number of previous tool in DBW (n+42) / Número de búfer de la herramienta previa en DBW (n+42)
   // // TIF[8].OldTinDBW42 : Puffernummer des vorherigen Werkzeugs in DBW (n+42) / Buffer number of previous tool in DBW (n+42) / Número de búfer de la herramienta previa en DBW (n+42)
   // // TIF[9].OldTinDBW42 : Puffernummer des vorherigen Werkzeugs in DBW (n+42) / Buffer number of previous tool in DBW (n+42) / Número de búfer de la herramienta previa en DBW (n+42)
   // // TIF[10].OldTinDBW42 : Puffernummer des vorherigen Werkzeugs in DBW (n+42) / Buffer number of previous tool in DBW (n+42) / Número de búfer de la herramienta previa en DBW (n+42)
   // // TIF[11].OldTinDBW42 : Puffernummer des vorherigen Werkzeugs in DBW (n+42) / Buffer number of previous tool in DBW (n+42) / Número de búfer de la herramienta previa en DBW (n+42)
   // // TIF[12].OldTinDBW42 : Puffernummer des vorherigen Werkzeugs in DBW (n+42) / Buffer number of previous tool in DBW (n+42) / Número de búfer de la herramienta previa en DBW (n+42)
   // // TIF[13].OldTinDBW42 : Puffernummer des vorherigen Werkzeugs in DBW (n+42) / Buffer number of previous tool in DBW (n+42) / Número de búfer de la herramienta previa en DBW (n+42)
   // // TIF[14].OldTinDBW42 : Puffernummer des vorherigen Werkzeugs in DBW (n+42) / Buffer number of previous tool in DBW (n+42) / Número de búfer de la herramienta previa en DBW (n+42)
   // // TIF[15].OldTinDBW42 : Puffernummer des vorherigen Werkzeugs in DBW (n+42) / Buffer number of previous tool in DBW (n+42) / Número de búfer de la herramienta previa en DBW (n+42)
   // // TIF[16].OldTinDBW42 : Puffernummer des vorherigen Werkzeugs in DBW (n+42) / Buffer number of previous tool in DBW (n+42) / Número de búfer de la herramienta previa en DBW (n+42)
   // // TIF[2].ManTIn : Handwerkzeug manuell in Spindel laden / Load hand tool in spindle manually / Cargar a mano herramienta manual en cabezal
   // // TIF[3].ManTIn : Handwerkzeug manuell in Spindel laden / Load hand tool in spindle manually / Cargar a mano herramienta manual en cabezal
   // // TIF[4].ManTIn : Handwerkzeug manuell in Spindel laden / Load hand tool in spindle manually / Cargar a mano herramienta manual en cabezal
   // // TIF[5].ManTIn : Handwerkzeug manuell in Spindel laden / Load hand tool in spindle manually / Cargar a mano herramienta manual en cabezal
   // // TIF[6].ManTIn : Handwerkzeug manuell in Spindel laden / Load hand tool in spindle manually / Cargar a mano herramienta manual en cabezal
   // // TIF[7].ManTIn : Handwerkzeug manuell in Spindel laden / Load hand tool in spindle manually / Cargar a mano herramienta manual en cabezal
   // // TIF[8].ManTIn : Handwerkzeug manuell in Spindel laden / Load hand tool in spindle manually / Cargar a mano herramienta manual en cabezal
   // // TIF[9].ManTIn : Handwerkzeug manuell in Spindel laden / Load hand tool in spindle manually / Cargar a mano herramienta manual en cabezal
   // // TIF[10].ManTIn : Handwerkzeug manuell in Spindel laden / Load hand tool in spindle manually / Cargar a mano herramienta manual en cabezal
   // // TIF[11].ManTIn : Handwerkzeug manuell in Spindel laden / Load hand tool in spindle manually / Cargar a mano herramienta manual en cabezal
   // // TIF[12].ManTIn : Handwerkzeug manuell in Spindel laden / Load hand tool in spindle manually / Cargar a mano herramienta manual en cabezal
   // // TIF[13].ManTIn : Handwerkzeug manuell in Spindel laden / Load hand tool in spindle manually / Cargar a mano herramienta manual en cabezal
   // // TIF[14].ManTIn : Handwerkzeug manuell in Spindel laden / Load hand tool in spindle manually / Cargar a mano herramienta manual en cabezal
   // // TIF[15].ManTIn : Handwerkzeug manuell in Spindel laden / Load hand tool in spindle manually / Cargar a mano herramienta manual en cabezal
   // // TIF[16].ManTIn : Handwerkzeug manuell in Spindel laden / Load hand tool in spindle manually / Cargar a mano herramienta manual en cabezal
   // // TIF[2].ManTOut : Handwerkzeug manuell aus Spindel entladen / Unload hand tool from spindle manually / Descargar a mano herramienta manual del cabezal
   // // TIF[3].ManTOut : Handwerkzeug manuell aus Spindel entladen / Unload hand tool from spindle manually / Descargar a mano herramienta manual del cabezal
   // // TIF[4].ManTOut : Handwerkzeug manuell aus Spindel entladen / Unload hand tool from spindle manually / Descargar a mano herramienta manual del cabezal
   // // TIF[5].ManTOut : Handwerkzeug manuell aus Spindel entladen / Unload hand tool from spindle manually / Descargar a mano herramienta manual del cabezal
   // // TIF[6].ManTOut : Handwerkzeug manuell aus Spindel entladen / Unload hand tool from spindle manually / Descargar a mano herramienta manual del cabezal
   // // TIF[7].ManTOut : Handwerkzeug manuell aus Spindel entladen / Unload hand tool from spindle manually / Descargar a mano herramienta manual del cabezal
   // // TIF[8].ManTOut : Handwerkzeug manuell aus Spindel entladen / Unload hand tool from spindle manually / Descargar a mano herramienta manual del cabezal
   // // TIF[9].ManTOut : Handwerkzeug manuell aus Spindel entladen / Unload hand tool from spindle manually / Descargar a mano herramienta manual del cabezal
   // // TIF[10].ManTOut : Handwerkzeug manuell aus Spindel entladen / Unload hand tool from spindle manually / Descargar a mano herramienta manual del cabezal
   // // TIF[11].ManTOut : Handwerkzeug manuell aus Spindel entladen / Unload hand tool from spindle manually / Descargar a mano herramienta manual del cabezal
   // // TIF[12].ManTOut : Handwerkzeug manuell aus Spindel entladen / Unload hand tool from spindle manually / Descargar a mano herramienta manual del cabezal
   // // TIF[13].ManTOut : Handwerkzeug manuell aus Spindel entladen / Unload hand tool from spindle manually / Descargar a mano herramienta manual del cabezal
   // // TIF[14].ManTOut : Handwerkzeug manuell aus Spindel entladen / Unload hand tool from spindle manually / Descargar a mano herramienta manual del cabezal
   // // TIF[15].ManTOut : Handwerkzeug manuell aus Spindel entladen / Unload hand tool from spindle manually / Descargar a mano herramienta manual del cabezal
   // // TIF[16].ManTOut : Handwerkzeug manuell aus Spindel entladen / Unload hand tool from spindle manually / Descargar a mano herramienta manual del cabezal
   // // TIF[2].SpiTRSpi : Spindelwerkzeug verbleibt in der Spindel / Spindle tool remains in spindle / Herramienta del cabezal permanece en el cabezal
   // // TIF[3].SpiTRSpi : Spindelwerkzeug verbleibt in der Spindel / Spindle tool remains in spindle / Herramienta del cabezal permanece en el cabezal
   // // TIF[4].SpiTRSpi : Spindelwerkzeug verbleibt in der Spindel / Spindle tool remains in spindle / Herramienta del cabezal permanece en el cabezal
   // // TIF[5].SpiTRSpi : Spindelwerkzeug verbleibt in der Spindel / Spindle tool remains in spindle / Herramienta del cabezal permanece en el cabezal
   // // TIF[6].SpiTRSpi : Spindelwerkzeug verbleibt in der Spindel / Spindle tool remains in spindle / Herramienta del cabezal permanece en el cabezal
   // // TIF[7].SpiTRSpi : Spindelwerkzeug verbleibt in der Spindel / Spindle tool remains in spindle / Herramienta del cabezal permanece en el cabezal
   // // TIF[8].SpiTRSpi : Spindelwerkzeug verbleibt in der Spindel / Spindle tool remains in spindle / Herramienta del cabezal permanece en el cabezal
   // // TIF[9].SpiTRSpi : Spindelwerkzeug verbleibt in der Spindel / Spindle tool remains in spindle / Herramienta del cabezal permanece en el cabezal
   // // TIF[10].SpiTRSpi : Spindelwerkzeug verbleibt in der Spindel / Spindle tool remains in spindle / Herramienta del cabezal permanece en el cabezal
   // // TIF[11].SpiTRSpi : Spindelwerkzeug verbleibt in der Spindel / Spindle tool remains in spindle / Herramienta del cabezal permanece en el cabezal
   // // TIF[12].SpiTRSpi : Spindelwerkzeug verbleibt in der Spindel / Spindle tool remains in spindle / Herramienta del cabezal permanece en el cabezal
   // // TIF[13].SpiTRSpi : Spindelwerkzeug verbleibt in der Spindel / Spindle tool remains in spindle / Herramienta del cabezal permanece en el cabezal
   // // TIF[14].SpiTRSpi : Spindelwerkzeug verbleibt in der Spindel / Spindle tool remains in spindle / Herramienta del cabezal permanece en el cabezal
   // // TIF[15].SpiTRSpi : Spindelwerkzeug verbleibt in der Spindel / Spindle tool remains in spindle / Herramienta del cabezal permanece en el cabezal
   // // TIF[16].SpiTRSpi : Spindelwerkzeug verbleibt in der Spindel / Spindle tool remains in spindle / Herramienta del cabezal permanece en el cabezal
   // // TIF[2].PerfStatusError : Negative Quittung / Negative acknowledge / Confirmación negativa
   // // TIF[3].PerfStatusError : Negative Quittung / Negative acknowledge / Confirmación negativa
   // // TIF[4].PerfStatusError : Negative Quittung / Negative acknowledge / Confirmación negativa
   // // TIF[5].PerfStatusError : Negative Quittung / Negative acknowledge / Confirmación negativa
   // // TIF[6].PerfStatusError : Negative Quittung / Negative acknowledge / Confirmación negativa
   // // TIF[7].PerfStatusError : Negative Quittung / Negative acknowledge / Confirmación negativa
   // // TIF[8].PerfStatusError : Negative Quittung / Negative acknowledge / Confirmación negativa
   // // TIF[9].PerfStatusError : Negative Quittung / Negative acknowledge / Confirmación negativa
   // // TIF[10].PerfStatusError : Negative Quittung / Negative acknowledge / Confirmación negativa
   // // TIF[11].PerfStatusError : Negative Quittung / Negative acknowledge / Confirmación negativa
   // // TIF[12].PerfStatusError : Negative Quittung / Negative acknowledge / Confirmación negativa
   // // TIF[13].PerfStatusError : Negative Quittung / Negative acknowledge / Confirmación negativa
   // // TIF[14].PerfStatusError : Negative Quittung / Negative acknowledge / Confirmación negativa
   // // TIF[15].PerfStatusError : Negative Quittung / Negative acknowledge / Confirmación negativa
   // // TIF[16].PerfStatusError : Negative Quittung / Negative acknowledge / Confirmación negativa
   // // TIF[2].n1_1 : Reserviert / Reserved / Reservado
   // // TIF[3].n1_1 : Reserviert / Reserved / Reservado
   // // TIF[4].n1_1 : Reserviert / Reserved / Reservado
   // // TIF[5].n1_1 : Reserviert / Reserved / Reservado
   // // TIF[6].n1_1 : Reserviert / Reserved / Reservado
   // // TIF[7].n1_1 : Reserviert / Reserved / Reservado
   // // TIF[8].n1_1 : Reserviert / Reserved / Reservado
   // // TIF[9].n1_1 : Reserviert / Reserved / Reservado
   // // TIF[10].n1_1 : Reserviert / Reserved / Reservado
   // // TIF[11].n1_1 : Reserviert / Reserved / Reservado
   // // TIF[12].n1_1 : Reserviert / Reserved / Reservado
   // // TIF[13].n1_1 : Reserviert / Reserved / Reservado
   // // TIF[14].n1_1 : Reserviert / Reserved / Reservado
   // // TIF[15].n1_1 : Reserviert / Reserved / Reservado
   // // TIF[16].n1_1 : Reserviert / Reserved / Reservado
   // // TIF[2].n1_2 : Reserviert / Reserved / Reservado
   // // TIF[3].n1_2 : Reserviert / Reserved / Reservado
   // // TIF[4].n1_2 : Reserviert / Reserved / Reservado
   // // TIF[5].n1_2 : Reserviert / Reserved / Reservado
   // // TIF[6].n1_2 : Reserviert / Reserved / Reservado
   // // TIF[7].n1_2 : Reserviert / Reserved / Reservado
   // // TIF[8].n1_2 : Reserviert / Reserved / Reservado
   // // TIF[9].n1_2 : Reserviert / Reserved / Reservado
   // // TIF[10].n1_2 : Reserviert / Reserved / Reservado
   // // TIF[11].n1_2 : Reserviert / Reserved / Reservado
   // // TIF[12].n1_2 : Reserviert / Reserved / Reservado
   // // TIF[13].n1_2 : Reserviert / Reserved / Reservado
   // // TIF[14].n1_2 : Reserviert / Reserved / Reservado
   // // TIF[15].n1_2 : Reserviert / Reserved / Reservado
   // // TIF[16].n1_2 : Reserviert / Reserved / Reservado
   // // TIF[2].n1_3 : Reserviert / Reserved / Reservado
   // // TIF[3].n1_3 : Reserviert / Reserved / Reservado
   // // TIF[4].n1_3 : Reserviert / Reserved / Reservado
   // // TIF[5].n1_3 : Reserviert / Reserved / Reservado
   // // TIF[6].n1_3 : Reserviert / Reserved / Reservado
   // // TIF[7].n1_3 : Reserviert / Reserved / Reservado
   // // TIF[8].n1_3 : Reserviert / Reserved / Reservado
   // // TIF[9].n1_3 : Reserviert / Reserved / Reservado
   // // TIF[10].n1_3 : Reserviert / Reserved / Reservado
   // // TIF[11].n1_3 : Reserviert / Reserved / Reservado
   // // TIF[12].n1_3 : Reserviert / Reserved / Reservado
   // // TIF[13].n1_3 : Reserviert / Reserved / Reservado
   // // TIF[14].n1_3 : Reserviert / Reserved / Reservado
   // // TIF[15].n1_3 : Reserviert / Reserved / Reservado
   // // TIF[16].n1_3 : Reserviert / Reserved / Reservado
   // // TIF[2].n1_4 : Reserviert / Reserved / Reservado
   // // TIF[3].n1_4 : Reserviert / Reserved / Reservado
   // // TIF[4].n1_4 : Reserviert / Reserved / Reservado
   // // TIF[5].n1_4 : Reserviert / Reserved / Reservado
   // // TIF[6].n1_4 : Reserviert / Reserved / Reservado
   // // TIF[7].n1_4 : Reserviert / Reserved / Reservado
   // // TIF[8].n1_4 : Reserviert / Reserved / Reservado
   // // TIF[9].n1_4 : Reserviert / Reserved / Reservado
   // // TIF[10].n1_4 : Reserviert / Reserved / Reservado
   // // TIF[11].n1_4 : Reserviert / Reserved / Reservado
   // // TIF[12].n1_4 : Reserviert / Reserved / Reservado
   // // TIF[13].n1_4 : Reserviert / Reserved / Reservado
   // // TIF[14].n1_4 : Reserviert / Reserved / Reservado
   // // TIF[15].n1_4 : Reserviert / Reserved / Reservado
   // // TIF[16].n1_4 : Reserviert / Reserved / Reservado
   // // TIF[2].n1_5 : Reserviert / Reserved / Reservado
   // // TIF[3].n1_5 : Reserviert / Reserved / Reservado
   // // TIF[4].n1_5 : Reserviert / Reserved / Reservado
   // // TIF[5].n1_5 : Reserviert / Reserved / Reservado
   // // TIF[6].n1_5 : Reserviert / Reserved / Reservado
   // // TIF[7].n1_5 : Reserviert / Reserved / Reservado
   // // TIF[8].n1_5 : Reserviert / Reserved / Reservado
   // // TIF[9].n1_5 : Reserviert / Reserved / Reservado
   // // TIF[10].n1_5 : Reserviert / Reserved / Reservado
   // // TIF[11].n1_5 : Reserviert / Reserved / Reservado
   // // TIF[12].n1_5 : Reserviert / Reserved / Reservado
   // // TIF[13].n1_5 : Reserviert / Reserved / Reservado
   // // TIF[14].n1_5 : Reserviert / Reserved / Reservado
   // // TIF[15].n1_5 : Reserviert / Reserved / Reservado
   // // TIF[16].n1_5 : Reserviert / Reserved / Reservado
   // // TIF[2].n1_6 : Reserviert / Reserved / Reservado
   // // TIF[3].n1_6 : Reserviert / Reserved / Reservado
   // // TIF[4].n1_6 : Reserviert / Reserved / Reservado
   // // TIF[5].n1_6 : Reserviert / Reserved / Reservado
   // // TIF[6].n1_6 : Reserviert / Reserved / Reservado
   // // TIF[7].n1_6 : Reserviert / Reserved / Reservado
   // // TIF[8].n1_6 : Reserviert / Reserved / Reservado
   // // TIF[9].n1_6 : Reserviert / Reserved / Reservado
   // // TIF[10].n1_6 : Reserviert / Reserved / Reservado
   // // TIF[11].n1_6 : Reserviert / Reserved / Reservado
   // // TIF[12].n1_6 : Reserviert / Reserved / Reservado
   // // TIF[13].n1_6 : Reserviert / Reserved / Reservado
   // // TIF[14].n1_6 : Reserviert / Reserved / Reservado
   // // TIF[15].n1_6 : Reserviert / Reserved / Reservado
   // // TIF[16].n1_6 : Reserviert / Reserved / Reservado
   // // TIF[2].DataInDB1072 : Multitool-Daten gespeichert in DB1072 / Multitool data stored in DB1072 / Datos Multitool guardados en DB1072
   // // TIF[3].DataInDB1072 : Multitool-Daten gespeichert in DB1072 / Multitool data stored in DB1072 / Datos Multitool guardados en DB1072
   // // TIF[4].DataInDB1072 : Multitool-Daten gespeichert in DB1072 / Multitool data stored in DB1072 / Datos Multitool guardados en DB1072
   // // TIF[5].DataInDB1072 : Multitool-Daten gespeichert in DB1072 / Multitool data stored in DB1072 / Datos Multitool guardados en DB1072
   // // TIF[6].DataInDB1072 : Multitool-Daten gespeichert in DB1072 / Multitool data stored in DB1072 / Datos Multitool guardados en DB1072
   // // TIF[7].DataInDB1072 : Multitool-Daten gespeichert in DB1072 / Multitool data stored in DB1072 / Datos Multitool guardados en DB1072
   // // TIF[8].DataInDB1072 : Multitool-Daten gespeichert in DB1072 / Multitool data stored in DB1072 / Datos Multitool guardados en DB1072
   // // TIF[9].DataInDB1072 : Multitool-Daten gespeichert in DB1072 / Multitool data stored in DB1072 / Datos Multitool guardados en DB1072
   // // TIF[10].DataInDB1072 : Multitool-Daten gespeichert in DB1072 / Multitool data stored in DB1072 / Datos Multitool guardados en DB1072
   // // TIF[11].DataInDB1072 : Multitool-Daten gespeichert in DB1072 / Multitool data stored in DB1072 / Datos Multitool guardados en DB1072
   // // TIF[12].DataInDB1072 : Multitool-Daten gespeichert in DB1072 / Multitool data stored in DB1072 / Datos Multitool guardados en DB1072
   // // TIF[13].DataInDB1072 : Multitool-Daten gespeichert in DB1072 / Multitool data stored in DB1072 / Datos Multitool guardados en DB1072
   // // TIF[14].DataInDB1072 : Multitool-Daten gespeichert in DB1072 / Multitool data stored in DB1072 / Datos Multitool guardados en DB1072
   // // TIF[15].DataInDB1072 : Multitool-Daten gespeichert in DB1072 / Multitool data stored in DB1072 / Datos Multitool guardados en DB1072
   // // TIF[16].DataInDB1072 : Multitool-Daten gespeichert in DB1072 / Multitool data stored in DB1072 / Datos Multitool guardados en DB1072
   // // TIF[2].Channel : Zugeordneter Kanal / Assigned channel / Canal asignado
   // // TIF[3].Channel : Zugeordneter Kanal / Assigned channel / Canal asignado
   // // TIF[4].Channel : Zugeordneter Kanal / Assigned channel / Canal asignado
   // // TIF[5].Channel : Zugeordneter Kanal / Assigned channel / Canal asignado
   // // TIF[6].Channel : Zugeordneter Kanal / Assigned channel / Canal asignado
   // // TIF[7].Channel : Zugeordneter Kanal / Assigned channel / Canal asignado
   // // TIF[8].Channel : Zugeordneter Kanal / Assigned channel / Canal asignado
   // // TIF[9].Channel : Zugeordneter Kanal / Assigned channel / Canal asignado
   // // TIF[10].Channel : Zugeordneter Kanal / Assigned channel / Canal asignado
   // // TIF[11].Channel : Zugeordneter Kanal / Assigned channel / Canal asignado
   // // TIF[12].Channel : Zugeordneter Kanal / Assigned channel / Canal asignado
   // // TIF[13].Channel : Zugeordneter Kanal / Assigned channel / Canal asignado
   // // TIF[14].Channel : Zugeordneter Kanal / Assigned channel / Canal asignado
   // // TIF[15].Channel : Zugeordneter Kanal / Assigned channel / Canal asignado
   // // TIF[16].Channel : Zugeordneter Kanal / Assigned channel / Canal asignado
   // // TIF[2].TMNo : Werkzeug-Verwaltungsnummer / Tool management number / Número de gestión de herramientas
   // // TIF[3].TMNo : Werkzeug-Verwaltungsnummer / Tool management number / Número de gestión de herramientas
   // // TIF[4].TMNo : Werkzeug-Verwaltungsnummer / Tool management number / Número de gestión de herramientas
   // // TIF[5].TMNo : Werkzeug-Verwaltungsnummer / Tool management number / Número de gestión de herramientas
   // // TIF[6].TMNo : Werkzeug-Verwaltungsnummer / Tool management number / Número de gestión de herramientas
   // // TIF[7].TMNo : Werkzeug-Verwaltungsnummer / Tool management number / Número de gestión de herramientas
   // // TIF[8].TMNo : Werkzeug-Verwaltungsnummer / Tool management number / Número de gestión de herramientas
   // // TIF[9].TMNo : Werkzeug-Verwaltungsnummer / Tool management number / Número de gestión de herramientas
   // // TIF[10].TMNo : Werkzeug-Verwaltungsnummer / Tool management number / Número de gestión de herramientas
   // // TIF[11].TMNo : Werkzeug-Verwaltungsnummer / Tool management number / Número de gestión de herramientas
   // // TIF[12].TMNo : Werkzeug-Verwaltungsnummer / Tool management number / Número de gestión de herramientas
   // // TIF[13].TMNo : Werkzeug-Verwaltungsnummer / Tool management number / Número de gestión de herramientas
   // // TIF[14].TMNo : Werkzeug-Verwaltungsnummer / Tool management number / Número de gestión de herramientas
   // // TIF[15].TMNo : Werkzeug-Verwaltungsnummer / Tool management number / Número de gestión de herramientas
   // // TIF[16].TMNo : Werkzeug-Verwaltungsnummer / Tool management number / Número de gestión de herramientas
   // // TIF[2].VdiTcp0 : Freie Anwendervariable 0 / User parameter 0 / Parámetro de usuario 0
   // // TIF[3].VdiTcp0 : Freie Anwendervariable 0 / User parameter 0 / Parámetro de usuario 0
   // // TIF[4].VdiTcp0 : Freie Anwendervariable 0 / User parameter 0 / Parámetro de usuario 0
   // // TIF[5].VdiTcp0 : Freie Anwendervariable 0 / User parameter 0 / Parámetro de usuario 0
   // // TIF[6].VdiTcp0 : Freie Anwendervariable 0 / User parameter 0 / Parámetro de usuario 0
   // // TIF[7].VdiTcp0 : Freie Anwendervariable 0 / User parameter 0 / Parámetro de usuario 0
   // // TIF[8].VdiTcp0 : Freie Anwendervariable 0 / User parameter 0 / Parámetro de usuario 0
   // // TIF[9].VdiTcp0 : Freie Anwendervariable 0 / User parameter 0 / Parámetro de usuario 0
   // // TIF[10].VdiTcp0 : Freie Anwendervariable 0 / User parameter 0 / Parámetro de usuario 0
   // // TIF[11].VdiTcp0 : Freie Anwendervariable 0 / User parameter 0 / Parámetro de usuario 0
   // // TIF[12].VdiTcp0 : Freie Anwendervariable 0 / User parameter 0 / Parámetro de usuario 0
   // // TIF[13].VdiTcp0 : Freie Anwendervariable 0 / User parameter 0 / Parámetro de usuario 0
   // // TIF[14].VdiTcp0 : Freie Anwendervariable 0 / User parameter 0 / Parámetro de usuario 0
   // // TIF[15].VdiTcp0 : Freie Anwendervariable 0 / User parameter 0 / Parámetro de usuario 0
   // // TIF[16].VdiTcp0 : Freie Anwendervariable 0 / User parameter 0 / Parámetro de usuario 0
   // // TIF[2].VdiTcp1 : Freie Anwendervariable 1 / User parameter 1 / Parámetro de usuario 1
   // // TIF[3].VdiTcp1 : Freie Anwendervariable 1 / User parameter 1 / Parámetro de usuario 1
   // // TIF[4].VdiTcp1 : Freie Anwendervariable 1 / User parameter 1 / Parámetro de usuario 1
   // // TIF[5].VdiTcp1 : Freie Anwendervariable 1 / User parameter 1 / Parámetro de usuario 1
   // // TIF[6].VdiTcp1 : Freie Anwendervariable 1 / User parameter 1 / Parámetro de usuario 1
   // // TIF[7].VdiTcp1 : Freie Anwendervariable 1 / User parameter 1 / Parámetro de usuario 1
   // // TIF[8].VdiTcp1 : Freie Anwendervariable 1 / User parameter 1 / Parámetro de usuario 1
   // // TIF[9].VdiTcp1 : Freie Anwendervariable 1 / User parameter 1 / Parámetro de usuario 1
   // // TIF[10].VdiTcp1 : Freie Anwendervariable 1 / User parameter 1 / Parámetro de usuario 1
   // // TIF[11].VdiTcp1 : Freie Anwendervariable 1 / User parameter 1 / Parámetro de usuario 1
   // // TIF[12].VdiTcp1 : Freie Anwendervariable 1 / User parameter 1 / Parámetro de usuario 1
   // // TIF[13].VdiTcp1 : Freie Anwendervariable 1 / User parameter 1 / Parámetro de usuario 1
   // // TIF[14].VdiTcp1 : Freie Anwendervariable 1 / User parameter 1 / Parámetro de usuario 1
   // // TIF[15].VdiTcp1 : Freie Anwendervariable 1 / User parameter 1 / Parámetro de usuario 1
   // // TIF[16].VdiTcp1 : Freie Anwendervariable 1 / User parameter 1 / Parámetro de usuario 1
   // // TIF[2].VdiTcp2 : Freie Anwendervariable 2 / User parameter 2 / Parámetro de usuario 2
   // // TIF[3].VdiTcp2 : Freie Anwendervariable 2 / User parameter 2 / Parámetro de usuario 2
   // // TIF[4].VdiTcp2 : Freie Anwendervariable 2 / User parameter 2 / Parámetro de usuario 2
   // // TIF[5].VdiTcp2 : Freie Anwendervariable 2 / User parameter 2 / Parámetro de usuario 2
   // // TIF[6].VdiTcp2 : Freie Anwendervariable 2 / User parameter 2 / Parámetro de usuario 2
   // // TIF[7].VdiTcp2 : Freie Anwendervariable 2 / User parameter 2 / Parámetro de usuario 2
   // // TIF[8].VdiTcp2 : Freie Anwendervariable 2 / User parameter 2 / Parámetro de usuario 2
   // // TIF[9].VdiTcp2 : Freie Anwendervariable 2 / User parameter 2 / Parámetro de usuario 2
   // // TIF[10].VdiTcp2 : Freie Anwendervariable 2 / User parameter 2 / Parámetro de usuario 2
   // // TIF[11].VdiTcp2 : Freie Anwendervariable 2 / User parameter 2 / Parámetro de usuario 2
   // // TIF[12].VdiTcp2 : Freie Anwendervariable 2 / User parameter 2 / Parámetro de usuario 2
   // // TIF[13].VdiTcp2 : Freie Anwendervariable 2 / User parameter 2 / Parámetro de usuario 2
   // // TIF[14].VdiTcp2 : Freie Anwendervariable 2 / User parameter 2 / Parámetro de usuario 2
   // // TIF[15].VdiTcp2 : Freie Anwendervariable 2 / User parameter 2 / Parámetro de usuario 2
   // // TIF[16].VdiTcp2 : Freie Anwendervariable 2 / User parameter 2 / Parámetro de usuario 2
   // // TIF[2].BufferIdent : Puffer-Identifikation (Festwert 9998) / Buffer identification (fixed value 9998) / Identificación de búfer (valor fijo 9998)
   // // TIF[3].BufferIdent : Puffer-Identifikation (Festwert 9998) / Buffer identification (fixed value 9998) / Identificación de búfer (valor fijo 9998)
   // // TIF[4].BufferIdent : Puffer-Identifikation (Festwert 9998) / Buffer identification (fixed value 9998) / Identificación de búfer (valor fijo 9998)
   // // TIF[5].BufferIdent : Puffer-Identifikation (Festwert 9998) / Buffer identification (fixed value 9998) / Identificación de búfer (valor fijo 9998)
   // // TIF[6].BufferIdent : Puffer-Identifikation (Festwert 9998) / Buffer identification (fixed value 9998) / Identificación de búfer (valor fijo 9998)
   // // TIF[7].BufferIdent : Puffer-Identifikation (Festwert 9998) / Buffer identification (fixed value 9998) / Identificación de búfer (valor fijo 9998)
   // // TIF[8].BufferIdent : Puffer-Identifikation (Festwert 9998) / Buffer identification (fixed value 9998) / Identificación de búfer (valor fijo 9998)
   // // TIF[9].BufferIdent : Puffer-Identifikation (Festwert 9998) / Buffer identification (fixed value 9998) / Identificación de búfer (valor fijo 9998)
   // // TIF[10].BufferIdent : Puffer-Identifikation (Festwert 9998) / Buffer identification (fixed value 9998) / Identificación de búfer (valor fijo 9998)
   // // TIF[11].BufferIdent : Puffer-Identifikation (Festwert 9998) / Buffer identification (fixed value 9998) / Identificación de búfer (valor fijo 9998)
   // // TIF[12].BufferIdent : Puffer-Identifikation (Festwert 9998) / Buffer identification (fixed value 9998) / Identificación de búfer (valor fijo 9998)
   // // TIF[13].BufferIdent : Puffer-Identifikation (Festwert 9998) / Buffer identification (fixed value 9998) / Identificación de búfer (valor fijo 9998)
   // // TIF[14].BufferIdent : Puffer-Identifikation (Festwert 9998) / Buffer identification (fixed value 9998) / Identificación de búfer (valor fijo 9998)
   // // TIF[15].BufferIdent : Puffer-Identifikation (Festwert 9998) / Buffer identification (fixed value 9998) / Identificación de búfer (valor fijo 9998)
   // // TIF[16].BufferIdent : Puffer-Identifikation (Festwert 9998) / Buffer identification (fixed value 9998) / Identificación de búfer (valor fijo 9998)
   // // TIF[2].BufferNo : Relativer Platz (Ziel) im Puffer / Relative location (target) in the buffer / Puesto relativo (destino) en el búfer
   // // TIF[3].BufferNo : Relativer Platz (Ziel) im Puffer / Relative location (target) in the buffer / Puesto relativo (destino) en el búfer
   // // TIF[4].BufferNo : Relativer Platz (Ziel) im Puffer / Relative location (target) in the buffer / Puesto relativo (destino) en el búfer
   // // TIF[5].BufferNo : Relativer Platz (Ziel) im Puffer / Relative location (target) in the buffer / Puesto relativo (destino) en el búfer
   // // TIF[6].BufferNo : Relativer Platz (Ziel) im Puffer / Relative location (target) in the buffer / Puesto relativo (destino) en el búfer
   // // TIF[7].BufferNo : Relativer Platz (Ziel) im Puffer / Relative location (target) in the buffer / Puesto relativo (destino) en el búfer
   // // TIF[8].BufferNo : Relativer Platz (Ziel) im Puffer / Relative location (target) in the buffer / Puesto relativo (destino) en el búfer
   // // TIF[9].BufferNo : Relativer Platz (Ziel) im Puffer / Relative location (target) in the buffer / Puesto relativo (destino) en el búfer
   // // TIF[10].BufferNo : Relativer Platz (Ziel) im Puffer / Relative location (target) in the buffer / Puesto relativo (destino) en el búfer
   // // TIF[11].BufferNo : Relativer Platz (Ziel) im Puffer / Relative location (target) in the buffer / Puesto relativo (destino) en el búfer
   // // TIF[12].BufferNo : Relativer Platz (Ziel) im Puffer / Relative location (target) in the buffer / Puesto relativo (destino) en el búfer
   // // TIF[13].BufferNo : Relativer Platz (Ziel) im Puffer / Relative location (target) in the buffer / Puesto relativo (destino) en el búfer
   // // TIF[14].BufferNo : Relativer Platz (Ziel) im Puffer / Relative location (target) in the buffer / Puesto relativo (destino) en el búfer
   // // TIF[15].BufferNo : Relativer Platz (Ziel) im Puffer / Relative location (target) in the buffer / Puesto relativo (destino) en el búfer
   // // TIF[16].BufferNo : Relativer Platz (Ziel) im Puffer / Relative location (target) in the buffer / Puesto relativo (destino) en el búfer
   // // TIF[2].SMag : Magazin-Nummer (Quelle) für neues Werkzeug / Magazine number (source) for new tool / Número de almacén (origen) para nueva herramienta
   // // TIF[3].SMag : Magazin-Nummer (Quelle) für neues Werkzeug / Magazine number (source) for new tool / Número de almacén (origen) para nueva herramienta
   // // TIF[4].SMag : Magazin-Nummer (Quelle) für neues Werkzeug / Magazine number (source) for new tool / Número de almacén (origen) para nueva herramienta
   // // TIF[5].SMag : Magazin-Nummer (Quelle) für neues Werkzeug / Magazine number (source) for new tool / Número de almacén (origen) para nueva herramienta
   // // TIF[6].SMag : Magazin-Nummer (Quelle) für neues Werkzeug / Magazine number (source) for new tool / Número de almacén (origen) para nueva herramienta
   // // TIF[7].SMag : Magazin-Nummer (Quelle) für neues Werkzeug / Magazine number (source) for new tool / Número de almacén (origen) para nueva herramienta
   // // TIF[8].SMag : Magazin-Nummer (Quelle) für neues Werkzeug / Magazine number (source) for new tool / Número de almacén (origen) para nueva herramienta
   // // TIF[9].SMag : Magazin-Nummer (Quelle) für neues Werkzeug / Magazine number (source) for new tool / Número de almacén (origen) para nueva herramienta
   // // TIF[10].SMag : Magazin-Nummer (Quelle) für neues Werkzeug / Magazine number (source) for new tool / Número de almacén (origen) para nueva herramienta
   // // TIF[11].SMag : Magazin-Nummer (Quelle) für neues Werkzeug / Magazine number (source) for new tool / Número de almacén (origen) para nueva herramienta
   // // TIF[12].SMag : Magazin-Nummer (Quelle) für neues Werkzeug / Magazine number (source) for new tool / Número de almacén (origen) para nueva herramienta
   // // TIF[13].SMag : Magazin-Nummer (Quelle) für neues Werkzeug / Magazine number (source) for new tool / Número de almacén (origen) para nueva herramienta
   // // TIF[14].SMag : Magazin-Nummer (Quelle) für neues Werkzeug / Magazine number (source) for new tool / Número de almacén (origen) para nueva herramienta
   // // TIF[15].SMag : Magazin-Nummer (Quelle) für neues Werkzeug / Magazine number (source) for new tool / Número de almacén (origen) para nueva herramienta
   // // TIF[16].SMag : Magazin-Nummer (Quelle) für neues Werkzeug / Magazine number (source) for new tool / Número de almacén (origen) para nueva herramienta
   // // TIF[2].SLoc : Platznummer (Quelle) für neues Werkzeug / Location number (source) for new tool / Número de puesto (origen) para nueva herramienta
   // // TIF[3].SLoc : Platznummer (Quelle) für neues Werkzeug / Location number (source) for new tool / Número de puesto (origen) para nueva herramienta
   // // TIF[4].SLoc : Platznummer (Quelle) für neues Werkzeug / Location number (source) for new tool / Número de puesto (origen) para nueva herramienta
   // // TIF[5].SLoc : Platznummer (Quelle) für neues Werkzeug / Location number (source) for new tool / Número de puesto (origen) para nueva herramienta
   // // TIF[6].SLoc : Platznummer (Quelle) für neues Werkzeug / Location number (source) for new tool / Número de puesto (origen) para nueva herramienta
   // // TIF[7].SLoc : Platznummer (Quelle) für neues Werkzeug / Location number (source) for new tool / Número de puesto (origen) para nueva herramienta
   // // TIF[8].SLoc : Platznummer (Quelle) für neues Werkzeug / Location number (source) for new tool / Número de puesto (origen) para nueva herramienta
   // // TIF[9].SLoc : Platznummer (Quelle) für neues Werkzeug / Location number (source) for new tool / Número de puesto (origen) para nueva herramienta
   // // TIF[10].SLoc : Platznummer (Quelle) für neues Werkzeug / Location number (source) for new tool / Número de puesto (origen) para nueva herramienta
   // // TIF[11].SLoc : Platznummer (Quelle) für neues Werkzeug / Location number (source) for new tool / Número de puesto (origen) para nueva herramienta
   // // TIF[12].SLoc : Platznummer (Quelle) für neues Werkzeug / Location number (source) for new tool / Número de puesto (origen) para nueva herramienta
   // // TIF[13].SLoc : Platznummer (Quelle) für neues Werkzeug / Location number (source) for new tool / Número de puesto (origen) para nueva herramienta
   // // TIF[14].SLoc : Platznummer (Quelle) für neues Werkzeug / Location number (source) for new tool / Número de puesto (origen) para nueva herramienta
   // // TIF[15].SLoc : Platznummer (Quelle) für neues Werkzeug / Location number (source) for new tool / Número de puesto (origen) para nueva herramienta
   // // TIF[16].SLoc : Platznummer (Quelle) für neues Werkzeug / Location number (source) for new tool / Número de puesto (origen) para nueva herramienta
   // // TIF[2].TMag : Magazin-Nummer (Ziel) für vorheriges Werkzeug / Magazine number (target) for previous tool / Número de almacén (destino) para herramienta previa
   // // TIF[3].TMag : Magazin-Nummer (Ziel) für vorheriges Werkzeug / Magazine number (target) for previous tool / Número de almacén (destino) para herramienta previa
   // // TIF[4].TMag : Magazin-Nummer (Ziel) für vorheriges Werkzeug / Magazine number (target) for previous tool / Número de almacén (destino) para herramienta previa
   // // TIF[5].TMag : Magazin-Nummer (Ziel) für vorheriges Werkzeug / Magazine number (target) for previous tool / Número de almacén (destino) para herramienta previa
   // // TIF[6].TMag : Magazin-Nummer (Ziel) für vorheriges Werkzeug / Magazine number (target) for previous tool / Número de almacén (destino) para herramienta previa
   // // TIF[7].TMag : Magazin-Nummer (Ziel) für vorheriges Werkzeug / Magazine number (target) for previous tool / Número de almacén (destino) para herramienta previa
   // // TIF[8].TMag : Magazin-Nummer (Ziel) für vorheriges Werkzeug / Magazine number (target) for previous tool / Número de almacén (destino) para herramienta previa
   // // TIF[9].TMag : Magazin-Nummer (Ziel) für vorheriges Werkzeug / Magazine number (target) for previous tool / Número de almacén (destino) para herramienta previa
   // // TIF[10].TMag : Magazin-Nummer (Ziel) für vorheriges Werkzeug / Magazine number (target) for previous tool / Número de almacén (destino) para herramienta previa
   // // TIF[11].TMag : Magazin-Nummer (Ziel) für vorheriges Werkzeug / Magazine number (target) for previous tool / Número de almacén (destino) para herramienta previa
   // // TIF[12].TMag : Magazin-Nummer (Ziel) für vorheriges Werkzeug / Magazine number (target) for previous tool / Número de almacén (destino) para herramienta previa
   // // TIF[13].TMag : Magazin-Nummer (Ziel) für vorheriges Werkzeug / Magazine number (target) for previous tool / Número de almacén (destino) para herramienta previa
   // // TIF[14].TMag : Magazin-Nummer (Ziel) für vorheriges Werkzeug / Magazine number (target) for previous tool / Número de almacén (destino) para herramienta previa
   // // TIF[15].TMag : Magazin-Nummer (Ziel) für vorheriges Werkzeug / Magazine number (target) for previous tool / Número de almacén (destino) para herramienta previa
   // // TIF[16].TMag : Magazin-Nummer (Ziel) für vorheriges Werkzeug / Magazine number (target) for previous tool / Número de almacén (destino) para herramienta previa
   // // TIF[2].TLoc : Platznummer (Ziel) für vorheriges Werkzeug / Location number (target) for previous tool / Número de puesto (destino) para herramienta previa
   // // TIF[3].TLoc : Platznummer (Ziel) für vorheriges Werkzeug / Location number (target) for previous tool / Número de puesto (destino) para herramienta previa
   // // TIF[4].TLoc : Platznummer (Ziel) für vorheriges Werkzeug / Location number (target) for previous tool / Número de puesto (destino) para herramienta previa
   // // TIF[5].TLoc : Platznummer (Ziel) für vorheriges Werkzeug / Location number (target) for previous tool / Número de puesto (destino) para herramienta previa
   // // TIF[6].TLoc : Platznummer (Ziel) für vorheriges Werkzeug / Location number (target) for previous tool / Número de puesto (destino) para herramienta previa
   // // TIF[7].TLoc : Platznummer (Ziel) für vorheriges Werkzeug / Location number (target) for previous tool / Número de puesto (destino) para herramienta previa
   // // TIF[8].TLoc : Platznummer (Ziel) für vorheriges Werkzeug / Location number (target) for previous tool / Número de puesto (destino) para herramienta previa
   // // TIF[9].TLoc : Platznummer (Ziel) für vorheriges Werkzeug / Location number (target) for previous tool / Número de puesto (destino) para herramienta previa
   // // TIF[10].TLoc : Platznummer (Ziel) für vorheriges Werkzeug / Location number (target) for previous tool / Número de puesto (destino) para herramienta previa
   // // TIF[11].TLoc : Platznummer (Ziel) für vorheriges Werkzeug / Location number (target) for previous tool / Número de puesto (destino) para herramienta previa
   // // TIF[12].TLoc : Platznummer (Ziel) für vorheriges Werkzeug / Location number (target) for previous tool / Número de puesto (destino) para herramienta previa
   // // TIF[13].TLoc : Platznummer (Ziel) für vorheriges Werkzeug / Location number (target) for previous tool / Número de puesto (destino) para herramienta previa
   // // TIF[14].TLoc : Platznummer (Ziel) für vorheriges Werkzeug / Location number (target) for previous tool / Número de puesto (destino) para herramienta previa
   // // TIF[15].TLoc : Platznummer (Ziel) für vorheriges Werkzeug / Location number (target) for previous tool / Número de puesto (destino) para herramienta previa
   // // TIF[16].TLoc : Platznummer (Ziel) für vorheriges Werkzeug / Location number (target) for previous tool / Número de puesto (destino) para herramienta previa
   // // TIF[2].LocType : Werkzeug neu: Platzart / Tool new: location type / Herramienta nueva: tipo de puesto
   // // TIF[3].LocType : Werkzeug neu: Platzart / Tool new: location type / Herramienta nueva: tipo de puesto
   // // TIF[4].LocType : Werkzeug neu: Platzart / Tool new: location type / Herramienta nueva: tipo de puesto
   // // TIF[5].LocType : Werkzeug neu: Platzart / Tool new: location type / Herramienta nueva: tipo de puesto
   // // TIF[6].LocType : Werkzeug neu: Platzart / Tool new: location type / Herramienta nueva: tipo de puesto
   // // TIF[7].LocType : Werkzeug neu: Platzart / Tool new: location type / Herramienta nueva: tipo de puesto
   // // TIF[8].LocType : Werkzeug neu: Platzart / Tool new: location type / Herramienta nueva: tipo de puesto
   // // TIF[9].LocType : Werkzeug neu: Platzart / Tool new: location type / Herramienta nueva: tipo de puesto
   // // TIF[10].LocType : Werkzeug neu: Platzart / Tool new: location type / Herramienta nueva: tipo de puesto
   // // TIF[11].LocType : Werkzeug neu: Platzart / Tool new: location type / Herramienta nueva: tipo de puesto
   // // TIF[12].LocType : Werkzeug neu: Platzart / Tool new: location type / Herramienta nueva: tipo de puesto
   // // TIF[13].LocType : Werkzeug neu: Platzart / Tool new: location type / Herramienta nueva: tipo de puesto
   // // TIF[14].LocType : Werkzeug neu: Platzart / Tool new: location type / Herramienta nueva: tipo de puesto
   // // TIF[15].LocType : Werkzeug neu: Platzart / Tool new: location type / Herramienta nueva: tipo de puesto
   // // TIF[16].LocType : Werkzeug neu: Platzart / Tool new: location type / Herramienta nueva: tipo de puesto
   // // TIF[2].SLeft : Werkeug neu: Größe links / Tool new: size left / Herramienta nueva: tamaño izquierda
   // // TIF[3].SLeft : Werkeug neu: Größe links / Tool new: size left / Herramienta nueva: tamaño izquierda
   // // TIF[4].SLeft : Werkeug neu: Größe links / Tool new: size left / Herramienta nueva: tamaño izquierda
   // // TIF[5].SLeft : Werkeug neu: Größe links / Tool new: size left / Herramienta nueva: tamaño izquierda
   // // TIF[6].SLeft : Werkeug neu: Größe links / Tool new: size left / Herramienta nueva: tamaño izquierda
   // // TIF[7].SLeft : Werkeug neu: Größe links / Tool new: size left / Herramienta nueva: tamaño izquierda
   // // TIF[8].SLeft : Werkeug neu: Größe links / Tool new: size left / Herramienta nueva: tamaño izquierda
   // // TIF[9].SLeft : Werkeug neu: Größe links / Tool new: size left / Herramienta nueva: tamaño izquierda
   // // TIF[10].SLeft : Werkeug neu: Größe links / Tool new: size left / Herramienta nueva: tamaño izquierda
   // // TIF[11].SLeft : Werkeug neu: Größe links / Tool new: size left / Herramienta nueva: tamaño izquierda
   // // TIF[12].SLeft : Werkeug neu: Größe links / Tool new: size left / Herramienta nueva: tamaño izquierda
   // // TIF[13].SLeft : Werkeug neu: Größe links / Tool new: size left / Herramienta nueva: tamaño izquierda
   // // TIF[14].SLeft : Werkeug neu: Größe links / Tool new: size left / Herramienta nueva: tamaño izquierda
   // // TIF[15].SLeft : Werkeug neu: Größe links / Tool new: size left / Herramienta nueva: tamaño izquierda
   // // TIF[16].SLeft : Werkeug neu: Größe links / Tool new: size left / Herramienta nueva: tamaño izquierda
   // // TIF[2].SRight : Werkeug neu: Größe rechts / Tool new: size right / Herramienta nueva: tamaño derecha
   // // TIF[3].SRight : Werkeug neu: Größe rechts / Tool new: size right / Herramienta nueva: tamaño derecha
   // // TIF[4].SRight : Werkeug neu: Größe rechts / Tool new: size right / Herramienta nueva: tamaño derecha
   // // TIF[5].SRight : Werkeug neu: Größe rechts / Tool new: size right / Herramienta nueva: tamaño derecha
   // // TIF[6].SRight : Werkeug neu: Größe rechts / Tool new: size right / Herramienta nueva: tamaño derecha
   // // TIF[7].SRight : Werkeug neu: Größe rechts / Tool new: size right / Herramienta nueva: tamaño derecha
   // // TIF[8].SRight : Werkeug neu: Größe rechts / Tool new: size right / Herramienta nueva: tamaño derecha
   // // TIF[9].SRight : Werkeug neu: Größe rechts / Tool new: size right / Herramienta nueva: tamaño derecha
   // // TIF[10].SRight : Werkeug neu: Größe rechts / Tool new: size right / Herramienta nueva: tamaño derecha
   // // TIF[11].SRight : Werkeug neu: Größe rechts / Tool new: size right / Herramienta nueva: tamaño derecha
   // // TIF[12].SRight : Werkeug neu: Größe rechts / Tool new: size right / Herramienta nueva: tamaño derecha
   // // TIF[13].SRight : Werkeug neu: Größe rechts / Tool new: size right / Herramienta nueva: tamaño derecha
   // // TIF[14].SRight : Werkeug neu: Größe rechts / Tool new: size right / Herramienta nueva: tamaño derecha
   // // TIF[15].SRight : Werkeug neu: Größe rechts / Tool new: size right / Herramienta nueva: tamaño derecha
   // // TIF[16].SRight : Werkeug neu: Größe rechts / Tool new: size right / Herramienta nueva: tamaño derecha
   // // TIF[2].STop : Werkeug neu: Größe oben / Tool new: size top / Herramienta nueva: tamaño arriba
   // // TIF[3].STop : Werkeug neu: Größe oben / Tool new: size top / Herramienta nueva: tamaño arriba
   // // TIF[4].STop : Werkeug neu: Größe oben / Tool new: size top / Herramienta nueva: tamaño arriba
   // // TIF[5].STop : Werkeug neu: Größe oben / Tool new: size top / Herramienta nueva: tamaño arriba
   // // TIF[6].STop : Werkeug neu: Größe oben / Tool new: size top / Herramienta nueva: tamaño arriba
   // // TIF[7].STop : Werkeug neu: Größe oben / Tool new: size top / Herramienta nueva: tamaño arriba
   // // TIF[8].STop : Werkeug neu: Größe oben / Tool new: size top / Herramienta nueva: tamaño arriba
   // // TIF[9].STop : Werkeug neu: Größe oben / Tool new: size top / Herramienta nueva: tamaño arriba
   // // TIF[10].STop : Werkeug neu: Größe oben / Tool new: size top / Herramienta nueva: tamaño arriba
   // // TIF[11].STop : Werkeug neu: Größe oben / Tool new: size top / Herramienta nueva: tamaño arriba
   // // TIF[12].STop : Werkeug neu: Größe oben / Tool new: size top / Herramienta nueva: tamaño arriba
   // // TIF[13].STop : Werkeug neu: Größe oben / Tool new: size top / Herramienta nueva: tamaño arriba
   // // TIF[14].STop : Werkeug neu: Größe oben / Tool new: size top / Herramienta nueva: tamaño arriba
   // // TIF[15].STop : Werkeug neu: Größe oben / Tool new: size top / Herramienta nueva: tamaño arriba
   // // TIF[16].STop : Werkeug neu: Größe oben / Tool new: size top / Herramienta nueva: tamaño arriba
   // // TIF[2].SBottom : Werkeug neu: Größe unten / Tool new: size bottom / Herramienta nueva: tamaño abajo
   // // TIF[3].SBottom : Werkeug neu: Größe unten / Tool new: size bottom / Herramienta nueva: tamaño abajo
   // // TIF[4].SBottom : Werkeug neu: Größe unten / Tool new: size bottom / Herramienta nueva: tamaño abajo
   // // TIF[5].SBottom : Werkeug neu: Größe unten / Tool new: size bottom / Herramienta nueva: tamaño abajo
   // // TIF[6].SBottom : Werkeug neu: Größe unten / Tool new: size bottom / Herramienta nueva: tamaño abajo
   // // TIF[7].SBottom : Werkeug neu: Größe unten / Tool new: size bottom / Herramienta nueva: tamaño abajo
   // // TIF[8].SBottom : Werkeug neu: Größe unten / Tool new: size bottom / Herramienta nueva: tamaño abajo
   // // TIF[9].SBottom : Werkeug neu: Größe unten / Tool new: size bottom / Herramienta nueva: tamaño abajo
   // // TIF[10].SBottom : Werkeug neu: Größe unten / Tool new: size bottom / Herramienta nueva: tamaño abajo
   // // TIF[11].SBottom : Werkeug neu: Größe unten / Tool new: size bottom / Herramienta nueva: tamaño abajo
   // // TIF[12].SBottom : Werkeug neu: Größe unten / Tool new: size bottom / Herramienta nueva: tamaño abajo
   // // TIF[13].SBottom : Werkeug neu: Größe unten / Tool new: size bottom / Herramienta nueva: tamaño abajo
